LIN {X 0,Y 340.752,Z 249.672,A -85,B 0,C 180,E1 -14239.386,E2 -14239.386} C_VEL
LIN {X 0,Y 341.112,Z 240.977,A -85,B 0,C 180,E1 -14243.046,E2 -14243.046} C_VEL
LIN {X 0,Y 341.383,Z 233.386,A -85,B 0,C 180,E1 -14246.271,E2 -14246.271} C_VEL
LIN {X 0,Y 341.787,Z 224.032,A -85,B 0,C 180,E1 -14250.272,E2 -14250.272} C_VEL
LIN {X 0,Y 342.168,Z 216.106,A -85,B 0,C 180,E1 -14253.681,E2 -14253.681} C_VEL
LIN {X 0,Y 342.261,Z 211.171,A -85,B 0,C 180,E1 -14255.819,E2 -14255.819} C_VEL
LIN {X 0,Y 341.512,Z 205.055,A -85,B 0,C 180,E1 -14258.554,E2 -14258.554} C_VEL
LIN {X 0,Y 340.75,Z 201.041,A -85,B 0,C 180,E1 -14260.45,E2 -14260.45} C_VEL
LIN {X 0,Y 340.658,Z 201.052,A -85,B 0,C 180,E1 -14263.772,E2 -14263.772} C_VEL
LIN {X 0,Y 340.704,Z 201.047,A -85,B 0,C 180,E1 -14267.954,E2 -14267.954} C_VEL
LIN {X 0,Y 340.725,Z 201.046,A -85,B 0,C 180,E1 -14271.77,E2 -14271.77} C_VEL
LIN {X 0,Y 340.727,Z 201.048,A -85,B 0,C 180,E1 -14275.595,E2 -14275.595} C_VEL
LIN {X 0,Y 340.674,Z 201.114,A -85,B 0,C 180,E1 -14278.779,E2 -14278.779} C_VEL
LIN {X 0,Y 340.81,Z 204.268,A -85,B 0,C 180,E1 -14281.685,E2 -14281.685} C_VEL
LIN {X 0,Y 340.762,Z 208.22,A -85,B 0,C 180,E1 -14285.159,E2 -14285.159} C_VEL
LIN {X 0,Y 340.627,Z 211.796,A -85,B 0,C 180,E1 -14288.197,E2 -14288.197} C_VEL
LIN {X 0,Y 340.62,Z 216.505,A -85,B 0,C 180,E1 -14291.97,E2 -14291.97} C_VEL
LIN {X 0,Y 340.593,Z 221.628,A -85,B 0,C 180,E1 -14295.786,E2 -14295.786} C_VEL
LIN {X 0,Y 343.415,Z 232.223,A -85,B 0,C 180,E1 -14296.441,E2 -14296.441} C_VEL
LIN {X 0,Y 345.261,Z 241.478,A -85,B 0,C 180,E1 -14297.204,E2 -14297.204} C_VEL
LIN {X 0,Y 345.073,Z 250.333,A -85,B 0,C 180,E1 -14298.081,E2 -14298.081} C_VEL
LIN {X 0,Y 344.549,Z 257.421,A -85,B 0,C 180,E1 -14298.974,E2 -14298.974} C_VEL
LIN {X 0,Y 343.928,Z 263.871,A -85,B 0,C 180,E1 -14299.996,E2 -14299.996} C_VEL
LIN {X 0,Y 343.24,Z 269.773,A -85,B 0,C 180,E1 -14301.165,E2 -14301.165} C_VEL
LIN {X 0,Y 342.737,Z 274.379,A -85,B 0,C 180,E1 -14302.339,E2 -14302.339} C_VEL
LIN {X 0,Y 342.185,Z 278.047,A -85,B 0,C 180,E1 -14303.512,E2 -14303.512} C_VEL
LIN {X 0,Y 341.789,Z 282.051,A -85,B 0,C 180,E1 -14305.281,E2 -14305.281} C_VEL
LIN {X 0,Y 341.323,Z 283.939,A -85,B 0,C 180,E1 -14306.457,E2 -14306.457} C_VEL
LIN {X 0,Y 341.219,Z 285.215,A -85,B 0,C 180,E1 -14307.638,E2 -14307.638} C_VEL
LIN {X 0,Y 341.059,Z 285.985,A -85,B 0,C 180,E1 -14308.818,E2 -14308.818} C_VEL
LIN {X 0,Y 340.993,Z 286.251,A -85,B 0,C 180,E1 -14309.998,E2 -14309.998} C_VEL
LIN {X 0,Y 341.056,Z 286.023,A -85,B 0,C 180,E1 -14311.179,E2 -14311.179} C_VEL
LIN {X 0,Y 341.213,Z 285.305,A -85,B 0,C 180,E1 -14312.359,E2 -14312.359} C_VEL
LIN {X 0,Y 341.32,Z 284.085,A -85,B 0,C 180,E1 -14313.54,E2 -14313.54} C_VEL
LIN {X 0,Y 342.009,Z 281.111,A -85,B 0,C 180,E1 -14315.304,E2 -14315.304} C_VEL
LIN {X 0,Y 342.279,Z 276.688,A -85,B 0,C 180,E1 -14317.075,E2 -14317.075} C_VEL
LIN {X 0,Y 342.822,Z 273.73,A -85,B 0,C 180,E1 -14317.952,E2 -14317.952} C_VEL
LIN {X 0,Y 343.198,Z 270.243,A -85,B 0,C 180,E1 -14318.833,E2 -14318.833} C_VEL
LIN {X 0,Y 343.922,Z 264.483,A -85,B 0,C 180,E1 -14320.001,E2 -14320.001} C_VEL
LIN {X 0,Y 344.435,Z 259.388,A -85,B 0,C 180,E1 -14320.849,E2 -14320.849} C_VEL
LIN {X 0,Y 344.905,Z 252.666,A -85,B 0,C 180,E1 -14321.756,E2 -14321.756} C_VEL
LIN {X 0,Y 345.44,Z 244.736,A -85,B 0,C 180,E1 -14322.602,E2 -14322.602} C_VEL
LIN {X 0,Y 345.523,Z 242.909,A -85,B 0,C 180,E1 -14322.763,E2 -14322.763} C_VEL
LIN {X 0,Y 343.767,Z 233.855,A -85,B 0,C 180,E1 -14323.547,E2 -14323.547} C_VEL
LIN {X 0,Y 341.183,Z 223.744,A -85,B 0,C 180,E1 -14324.209,E2 -14324.209} C_VEL
LIN {X 0,Y 340.594,Z 221.624,A -85,B 0,C 180,E1 -14324.335,E2 -14324.335} C_VEL
LIN {X 0,Y 340.626,Z 216.247,A -85,B 0,C 180,E1 -14328.359,E2 -14328.359} C_VEL
LIN {X 0,Y 340.65,Z 211.945,A -85,B 0,C 180,E1 -14331.812,E2 -14331.812} C_VEL
LIN {X 0,Y 340.771,Z 207.431,A -85,B 0,C 180,E1 -14335.663,E2 -14335.663} C_VEL
LIN {X 0,Y 340.815,Z 204.47,A -85,B 0,C 180,E1 -14338.311,E2 -14338.311} C_VEL
LIN {X 0,Y 340.696,Z 201.071,A -85,B 0,C 180,E1 -14341.388,E2 -14341.388} C_VEL
LIN {X 0,Y 340.714,Z 201.045,A -85,B 0,C 180,E1 -14345.277,E2 -14345.277} C_VEL
LIN {X 0,Y 340.707,Z 201.045,A -85,B 0,C 180,E1 -14348.385,E2 -14348.385} C_VEL
LIN {X 0,Y 340.693,Z 201.046,A -85,B 0,C 180,E1 -14352.044,E2 -14352.044} C_VEL
LIN {X 0,Y 340.655,Z 201.049,A -85,B 0,C 180,E1 -14353.428,E2 -14353.428} C_VEL
LIN {X 0,Y 339.988,Z 201.133,A -85,B 0,C 180,E1 -14354.413,E2 -14354.413} C_VEL
LIN {X 0,Y 337.121,Z 201.49,A -85,B 0,C 180,E1 -14356.017,E2 -14356.017} C_VEL
LIN {X 0,Y 334.701,Z 201.795,A -85,B 0,C 180,E1 -14357.315,E2 -14357.315} C_VEL
LIN {X 0,Y 333.681,Z 201.921,A -85,B 0,C 180,E1 -14358.32,E2 -14358.32} C_VEL
LIN {X 0,Y 333.607,Z 201.923,A -85,B 0,C 180,E1 -14358.66,E2 -14358.66} C_VEL
LIN {X 0,Y 333.645,Z 201.921,A -85,B 0,C 180,E1 -14362.348,E2 -14362.348} C_VEL
LIN {X 0,Y 333.666,Z 201.919,A -85,B 0,C 180,E1 -14365.34,E2 -14365.34} C_VEL
LIN {X 0,Y 333.691,Z 201.916,A -85,B 0,C 180,E1 -14369.637,E2 -14369.637} C_VEL
LIN {X 0,Y 333.735,Z 201.916,A -85,B 0,C 180,E1 -14372.4,E2 -14372.4} C_VEL
LIN {X 0,Y 333.717,Z 201.905,A -85,B 0,C 180,E1 -14375.09,E2 -14375.09} C_VEL
LIN {X 0,Y 333.672,Z 201.915,A -85,B 0,C 180,E1 -14379.018,E2 -14379.018} C_VEL
LIN {X 0,Y 333.784,Z 201.906,A -85,B 0,C 180,E1 -14381.589,E2 -14381.589} C_VEL
LIN {X 0,Y 333.797,Z 201.897,A -85,B 0,C 180,E1 -14385.576,E2 -14385.576} C_VEL
LIN {X 0,Y 333.823,Z 201.897,A -85,B 0,C 180,E1 -14389.078,E2 -14389.078} C_VEL
LIN {X 0,Y 333.994,Z 201.88,A -85,B 0,C 180,E1 -14392.747,E2 -14392.747} C_VEL
LIN {X 0,Y 333.797,Z 201.895,A -85,B 0,C 180,E1 -14395.169,E2 -14395.169} C_VEL
LIN {X 0,Y 334.095,Z 201.867,A -85,B 0,C 180,E1 -14397.589,E2 -14397.589} C_VEL
LIN {X 0,Y 334.235,Z 201.838,A -85,B 0,C 180,E1 -14400,E2 -14400} C_VEL
LIN {X 0,Y 334.092,Z 201.868,A -85,B 0,C 180,E1 -14402.411,E2 -14402.411} C_VEL
LIN {X 0,Y 334.012,Z 201.878,A -85,B 0,C 180,E1 -14407.253,E2 -14407.253} C_VEL
LIN {X 0,Y 333.822,Z 201.904,A -85,B 0,C 180,E1 -14410.922,E2 -14410.922} C_VEL
LIN {X 0,Y 333.797,Z 201.905,A -85,B 0,C 180,E1 -14414.635,E2 -14414.635} C_VEL
LIN {X 0,Y 333.712,Z 201.917,A -85,B 0,C 180,E1 -14418.618,E2 -14418.618} C_VEL
LIN {X 0,Y 333.64,Z 201.927,A -85,B 0,C 180,E1 -14422.282,E2 -14422.282} C_VEL
LIN {X 0,Y 333.648,Z 201.926,A -85,B 0,C 180,E1 -14425.079,E2 -14425.079} C_VEL
LIN {X 0,Y 333.64,Z 201.927,A -85,B 0,C 180,E1 -14428.979,E2 -14428.979} C_VEL
LIN {X 0,Y 333.634,Z 201.925,A -85,B 0,C 180,E1 -14432.588,E2 -14432.588} C_VEL
LIN {X 0,Y 333.666,Z 201.923,A -85,B 0,C 180,E1 -14436.14,E2 -14436.14} C_VEL
LIN {X 0,Y 333.611,Z 201.927,A -85,B 0,C 180,E1 -14439.197,E2 -14439.197} C_VEL
LIN {X 0,Y 333.621,Z 201.931,A -85,B 0,C 180,E1 -14442.501,E2 -14442.501} C_VEL
LIN {X 0,Y 333.608,Z 201.963,A -85,B 0,C 180,E1 -14445.143,E2 -14445.143} C_VEL
LIN {X 0,Y 335.798,Z 210.783,A -85,B 0,C 180,E1 -14448.891,E2 -14448.891} C_VEL
LIN {X 0,Y 337.805,Z 219.524,A -85,B 0,C 180,E1 -14452.24,E2 -14452.24} C_VEL
LIN {X 0,Y 339.708,Z 228.008,A -85,B 0,C 180,E1 -14455.259,E2 -14455.259} C_VEL
LIN {X 0,Y 340.958,Z 235.046,A -85,B 0,C 180,E1 -14457.595,E2 -14457.595} C_VEL
LIN {X 0,Y 338.442,Z 248.328,A -85,B 0,C 180,E1 -14461.473,E2 -14461.473} C_VEL
LIN {X 0,Y 336.139,Z 262.557,A -85,B 0,C 180,E1 -14465.613,E2 -14465.613} C_VEL
LIN {X 0,Y 334.245,Z 277.674,A -85,B 0,C 180,E1 -14470.043,E2 -14470.043} C_VEL
LIN {X 0,Y 335.25,Z 290.913,A -85,B 0,C 180,E1 -14470.623,E2 -14470.623} C_VEL
LIN {X 0,Y 336.597,Z 313.747,A -85,B 0,C 180,E1 -14472.065,E2 -14472.065} C_VEL
LIN {X 0,Y 336.521,Z 321.792,A -85,B 0,C 180,E1 -14472.688,E2 -14472.688} C_VEL
LIN {X 0,Y 335.458,Z 334.49,A -85,B 0,C 180,E1 -14473.885,E2 -14473.885} C_VEL
LIN {X 0,Y 334.585,Z 345.319,A -85,B 0,C 180,E1 -14475.186,E2 -14475.186} C_VEL
LIN {X 0,Y 333.812,Z 355.01,A -85,B 0,C 180,E1 -14476.611,E2 -14476.611} C_VEL
LIN {X 0,Y 333.237,Z 363.566,A -85,B 0,C 180,E1 -14478.135,E2 -14478.135} C_VEL
LIN {X 0,Y 332.682,Z 371.88,A -85,B 0,C 180,E1 -14479.965,E2 -14479.965} C_VEL
LIN {X 0,Y 332.422,Z 378.567,A -85,B 0,C 180,E1 -14481.797,E2 -14481.797} C_VEL
LIN {X 0,Y 332.288,Z 384.611,A -85,B 0,C 180,E1 -14483.931,E2 -14483.931} C_VEL
LIN {X 0,Y 332.272,Z 388.45,A -85,B 0,C 180,E1 -14485.756,E2 -14485.756} C_VEL
LIN {X 0,Y 332.413,Z 391.197,A -85,B 0,C 180,E1 -14487.578,E2 -14487.578} C_VEL
LIN {X 0,Y 332.392,Z 392.431,A -85,B 0,C 180,E1 -14488.79,E2 -14488.79} C_VEL
LIN {X 0,Y 332.398,Z 393.245,A -85,B 0,C 180,E1 -14490.002,E2 -14490.002} C_VEL
LIN {X 0,Y 332.364,Z 393.606,A -85,B 0,C 180,E1 -14491.213,E2 -14491.213} C_VEL
LIN {X 0,Y 332.207,Z 393.509,A -85,B 0,C 180,E1 -14492.427,E2 -14492.427} C_VEL
LIN {X 0,Y 332.156,Z 393.007,A -85,B 0,C 180,E1 -14493.641,E2 -14493.641} C_VEL
LIN {X 0,Y 332.142,Z 392.099,A -85,B 0,C 180,E1 -14494.857,E2 -14494.857} C_VEL
LIN {X 0,Y 332.153,Z 390.742,A -85,B 0,C 180,E1 -14496.074,E2 -14496.074} C_VEL
LIN {X 0,Y 332.362,Z 387.927,A -85,B 0,C 180,E1 -14497.902,E2 -14497.902} C_VEL
LIN {X 0,Y 332.773,Z 384.115,A -85,B 0,C 180,E1 -14499.729,E2 -14499.729} C_VEL
LIN {X 0,Y 333.487,Z 379.222,A -85,B 0,C 180,E1 -14501.55,E2 -14501.55} C_VEL
LIN {X 0,Y 334.831,Z 372.017,A -85,B 0,C 180,E1 -14503.66,E2 -14503.66} C_VEL
LIN {X 0,Y 336.173,Z 364.432,A -85,B 0,C 180,E1 -14505.461,E2 -14505.461} C_VEL
LIN {X 0,Y 337.605,Z 356.881,A -85,B 0,C 180,E1 -14506.946,E2 -14506.946} C_VEL
LIN {X 0,Y 339.904,Z 345.97,A -85,B 0,C 180,E1 -14508.694,E2 -14508.694} C_VEL
LIN {X 0,Y 342.101,Z 334.974,A -85,B 0,C 180,E1 -14510.129,E2 -14510.129} C_VEL
LIN {X 0,Y 343.964,Z 324.376,A -85,B 0,C 180,E1 -14511.266,E2 -14511.266} C_VEL
LIN {X 0,Y 345.101,Z 311.884,A -85,B 0,C 180,E1 -14512.459,E2 -14512.459} C_VEL
LIN {X 0,Y 345.075,Z 299.035,A -85,B 0,C 180,E1 -14513.58,E2 -14513.58} C_VEL
LIN {X 0,Y 343.453,Z 284.713,A -85,B 0,C 180,E1 -14514.796,E2 -14514.796} C_VEL
LIN {X 0,Y 341.202,Z 273.036,A -85,B 0,C 180,E1 -14515.877,E2 -14515.877} C_VEL
LIN {X 0,Y 341.429,Z 262.711,A -85,B 0,C 180,E1 -14517.734,E2 -14517.734} C_VEL
LIN {X 0,Y 342.068,Z 254.065,A -85,B 0,C 180,E1 -14519.546,E2 -14519.546} C_VEL
LIN {X 0,Y 343.381,Z 244.939,A -85,B 0,C 180,E1 -14521.806,E2 -14521.806} C_VEL
LIN {X 0,Y 344.103,Z 240.547,A -85,B 0,C 180,E1 -14523.134,E2 -14523.134} C_VEL
LIN {X 0,Y 343.908,Z 236.158,A -85,B 0,C 180,E1 -14525.172,E2 -14525.172} C_VEL
LIN {X 0,Y 343.989,Z 232.945,A -85,B 0,C 180,E1 -14527.174,E2 -14527.174} C_VEL
LIN {X 0,Y 344.239,Z 230.518,A -85,B 0,C 180,E1 -14529.266,E2 -14529.266} C_VEL
LIN {X 0,Y 344.234,Z 229.501,A -85,B 0,C 180,E1 -14530.939,E2 -14530.939} C_VEL
LIN {X 0,Y 343.907,Z 229.317,A -85,B 0,C 180,E1 -14532.635,E2 -14532.635} C_VEL
LIN {X 0,Y 343.51,Z 230.306,A -85,B 0,C 180,E1 -14535.923,E2 -14535.923} C_VEL
LIN {X 0,Y 343.392,Z 232.751,A -85,B 0,C 180,E1 -14539.225,E2 -14539.225} C_VEL
LIN {X 0,Y 343.344,Z 235.911,A -85,B 0,C 180,E1 -14542.115,E2 -14542.115} C_VEL
LIN {X 0,Y 343.1,Z 237.846,A -85,B 0,C 180,E1 -14543.556,E2 -14543.556} C_VEL
LIN {X 0,Y 341.056,Z 244.858,A -85,B 0,C 180,E1 -14547.66,E2 -14547.66} C_VEL
LIN {X 0,Y 339.549,Z 252.071,A -85,B 0,C 180,E1 -14551.572,E2 -14551.572} C_VEL
LIN {X 0,Y 338.917,Z 256.838,A -85,B 0,C 180,E1 -14553.975,E2 -14553.975} C_VEL
LIN {X 0,Y 343.148,Z 267.603,A -85,B 0,C 180,E1 -14555.465,E2 -14555.465} C_VEL
LIN {X 0,Y 346.448,Z 278.711,A -85,B 0,C 180,E1 -14556.923,E2 -14556.923} C_VEL
LIN {X 0,Y 347.886,Z 286.492,A -85,B 0,C 180,E1 -14557.908,E2 -14557.908} C_VEL
LIN {X 0,Y 347.59,Z 290.2,A -85,B 0,C 180,E1 -14558.273,E2 -14558.273} C_VEL
LIN {X 0,Y 345.38,Z 302.97,A -85,B 0,C 180,E1 -14559.606,E2 -14559.606} C_VEL
LIN {X 0,Y 343.032,Z 314.829,A -85,B 0,C 180,E1 -14561.175,E2 -14561.175} C_VEL
LIN {X 0,Y 340.728,Z 325.274,A -85,B 0,C 180,E1 -14562.907,E2 -14562.907} C_VEL
LIN {X 0,Y 338.756,Z 333.793,A -85,B 0,C 180,E1 -14564.662,E2 -14564.662} C_VEL
LIN {X 0,Y 337.117,Z 340.723,A -85,B 0,C 180,E1 -14566.436,E2 -14566.436} C_VEL
LIN {X 0,Y 335.629,Z 347.162,A -85,B 0,C 180,E1 -14568.526,E2 -14568.526} C_VEL
LIN {X 0,Y 334.586,Z 351.456,A -85,B 0,C 180,E1 -14570.326,E2 -14570.326} C_VEL
LIN {X 0,Y 334.005,Z 353.755,A -85,B 0,C 180,E1 -14571.53,E2 -14571.53} C_VEL
LIN {X 0,Y 333.364,Z 355.6,A -85,B 0,C 180,E1 -14572.733,E2 -14572.733} C_VEL
LIN {X 0,Y 332.998,Z 358.025,A -85,B 0,C 180,E1 -14575.157,E2 -14575.157} C_VEL
LIN {X 0,Y 332.712,Z 358.621,A -85,B 0,C 180,E1 -14576.367,E2 -14576.367} C_VEL
LIN {X 0,Y 332.318,Z 358.628,A -85,B 0,C 180,E1 -14578.788,E2 -14578.788} C_VEL
LIN {X 0,Y 332.22,Z 358.017,A -85,B 0,C 180,E1 -14580,E2 -14580} C_VEL
LIN {X 0,Y 332.192,Z 356.966,A -85,B 0,C 180,E1 -14581.212,E2 -14581.212} C_VEL
LIN {X 0,Y 332.19,Z 355.515,A -85,B 0,C 180,E1 -14582.425,E2 -14582.425} C_VEL
LIN {X 0,Y 332.318,Z 352.511,A -85,B 0,C 180,E1 -14584.245,E2 -14584.245} C_VEL
LIN {X 0,Y 332.458,Z 348.452,A -85,B 0,C 180,E1 -14586.067,E2 -14586.067} C_VEL
LIN {X 0,Y 332.843,Z 342.227,A -85,B 0,C 180,E1 -14588.194,E2 -14588.194} C_VEL
LIN {X 0,Y 333.379,Z 335.446,A -85,B 0,C 180,E1 -14590.016,E2 -14590.016} C_VEL
LIN {X 0,Y 334.013,Z 327.092,A -85,B 0,C 180,E1 -14591.838,E2 -14591.838} C_VEL
LIN {X 0,Y 334.942,Z 316.687,A -85,B 0,C 180,E1 -14593.654,E2 -14593.654} C_VEL
LIN {X 0,Y 335.846,Z 305.991,A -85,B 0,C 180,E1 -14595.164,E2 -14595.164} C_VEL
LIN {X 0,Y 336.612,Z 294.467,A -85,B 0,C 180,E1 -14596.481,E2 -14596.481} C_VEL
LIN {X 0,Y 337.485,Z 282.446,A -85,B 0,C 180,E1 -14597.575,E2 -14597.575} C_VEL
LIN {X 0,Y 337.858,Z 275.403,A -85,B 0,C 180,E1 -14598.103,E2 -14598.103} C_VEL
LIN {X 0,Y 335.673,Z 262.061,A -85,B 0,C 180,E1 -14599.003,E2 -14599.003} C_VEL
LIN {X 0,Y 333.741,Z 249.961,A -85,B 0,C 180,E1 -14599.633,E2 -14599.633} C_VEL
LIN {X 0,Y 334.135,Z 240.744,A -85,B 0,C 180,E1 -14603.556,E2 -14603.556} C_VEL
LIN {X 0,Y 334.468,Z 231.492,A -85,B 0,C 180,E1 -14607.534,E2 -14607.534} C_VEL
LIN {X 0,Y 334.959,Z 221.997,A -85,B 0,C 180,E1 -14611.638,E2 -14611.638} C_VEL
LIN {X 0,Y 335.281,Z 213.92,A -85,B 0,C 180,E1 -14615.163,E2 -14615.163} C_VEL
LIN {X 0,Y 334.916,Z 208.697,A -85,B 0,C 180,E1 -14617.485,E2 -14617.485} C_VEL
LIN {X 0,Y 333.707,Z 201.919,A -85,B 0,C 180,E1 -14620.644,E2 -14620.644} C_VEL
LIN {X 0,Y 333.599,Z 201.932,A -85,B 0,C 180,E1 -14624.25,E2 -14624.25} C_VEL
LIN {X 0,Y 333.647,Z 201.925,A -85,B 0,C 180,E1 -14627.618,E2 -14627.618} C_VEL
LIN {X 0,Y 333.645,Z 201.927,A -85,B 0,C 180,E1 -14631.204,E2 -14631.204} C_VEL
LIN {X 0,Y 333.678,Z 201.925,A -85,B 0,C 180,E1 -14633.86,E2 -14633.86} C_VEL
LIN {X 0,Y 333.638,Z 201.928,A -85,B 0,C 180,E1 -14637.415,E2 -14637.415} C_VEL
LIN {X 0,Y 333.689,Z 202.166,A -85,B 0,C 180,E1 -14638.581,E2 -14638.581} C_VEL
LIN {X 0,Y 333.797,Z 204.794,A -85,B 0,C 180,E1 -14641.035,E2 -14641.035} C_VEL
LIN {X 0,Y 333.765,Z 207.808,A -85,B 0,C 180,E1 -14643.755,E2 -14643.755} C_VEL
LIN {X 0,Y 333.692,Z 210.874,A -85,B 0,C 180,E1 -14646.41,E2 -14646.41} C_VEL
LIN {X 0,Y 333.578,Z 215.548,A -85,B 0,C 180,E1 -14650.298,E2 -14650.298} C_VEL
LIN {X 0,Y 333.556,Z 218.793,A -85,B 0,C 180,E1 -14652.842,E2 -14652.842} C_VEL
LIN {X 0,Y 333.553,Z 222.253,A -85,B 0,C 180,E1 -14655.411,E2 -14655.411} C_VEL
LIN {X 0,Y 336.552,Z 233.253,A -85,B 0,C 180,E1 -14656.124,E2 -14656.124} C_VEL
LIN {X 0,Y 338.447,Z 242.787,A -85,B 0,C 180,E1 -14656.939,E2 -14656.939} C_VEL
LIN {X 0,Y 338.237,Z 251.449,A -85,B 0,C 180,E1 -14657.829,E2 -14657.829} C_VEL
LIN {X 0,Y 337.667,Z 258.535,A -85,B 0,C 180,E1 -14658.746,E2 -14658.746} C_VEL
LIN {X 0,Y 337.022,Z 264.938,A -85,B 0,C 180,E1 -14659.789,E2 -14659.789} C_VEL
LIN {X 0,Y 336.299,Z 270.802,A -85,B 0,C 180,E1 -14660.981,E2 -14660.981} C_VEL
LIN {X 0,Y 335.775,Z 275.387,A -85,B 0,C 180,E1 -14662.179,E2 -14662.179} C_VEL
LIN {X 0,Y 335.203,Z 279.041,A -85,B 0,C 180,E1 -14663.377,E2 -14663.377} C_VEL
LIN {X 0,Y 334.789,Z 283.032,A -85,B 0,C 180,E1 -14665.182,E2 -14665.182} C_VEL
LIN {X 0,Y 334.311,Z 284.916,A -85,B 0,C 180,E1 -14666.383,E2 -14666.383} C_VEL
LIN {X 0,Y 334.199,Z 286.189,A -85,B 0,C 180,E1 -14667.588,E2 -14667.588} C_VEL
LIN {X 0,Y 334.034,Z 286.959,A -85,B 0,C 180,E1 -14668.793,E2 -14668.793} C_VEL
LIN {X 0,Y 333.966,Z 287.225,A -85,B 0,C 180,E1 -14669.998,E2 -14669.998} C_VEL
LIN {X 0,Y 334.031,Z 286.996,A -85,B 0,C 180,E1 -14671.204,E2 -14671.204} C_VEL
LIN {X 0,Y 334.193,Z 286.279,A -85,B 0,C 180,E1 -14672.409,E2 -14672.409} C_VEL
LIN {X 0,Y 334.308,Z 285.06,A -85,B 0,C 180,E1 -14673.614,E2 -14673.614} C_VEL
LIN {X 0,Y 335.014,Z 282.094,A -85,B 0,C 180,E1 -14675.415,E2 -14675.415} C_VEL
LIN {X 0,Y 335.304,Z 277.685,A -85,B 0,C 180,E1 -14677.223,E2 -14677.223} C_VEL
LIN {X 0,Y 335.865,Z 274.733,A -85,B 0,C 180,E1 -14678.118,E2 -14678.118} C_VEL
LIN {X 0,Y 336.259,Z 271.273,A -85,B 0,C 180,E1 -14679.017,E2 -14679.017} C_VEL
LIN {X 0,Y 337.018,Z 265.544,A -85,B 0,C 180,E1 -14680.208,E2 -14680.208} C_VEL
LIN {X 0,Y 337.558,Z 260.407,A -85,B 0,C 180,E1 -14681.085,E2 -14681.085} C_VEL
LIN {X 0,Y 338.047,Z 253.836,A -85,B 0,C 180,E1 -14681.998,E2 -14681.998} C_VEL
LIN {X 0,Y 338.595,Z 246.012,A -85,B 0,C 180,E1 -14682.861,E2 -14682.861} C_VEL
LIN {X 0,Y 338.415,Z 242.431,A -85,B 0,C 180,E1 -14683.204,E2 -14683.204} C_VEL
LIN {X 0,Y 336.365,Z 232.458,A -85,B 0,C 180,E1 -14684.046,E2 -14684.046} C_VEL
LIN {X 0,Y 333.581,Z 222.227,A -85,B 0,C 180,E1 -14684.721,E2 -14684.721} C_VEL
LIN {X 0,Y 333.605,Z 217.149,A -85,B 0,C 180,E1 -14688.556,E2 -14688.556} C_VEL
LIN {X 0,Y 333.639,Z 212.569,A -85,B 0,C 180,E1 -14692.28,E2 -14692.28} C_VEL
LIN {X 0,Y 333.755,Z 209.259,A -85,B 0,C 180,E1 -14695.113,E2 -14695.113} C_VEL
LIN {X 0,Y 333.847,Z 206.185,A -85,B 0,C 180,E1 -14697.85,E2 -14697.85} C_VEL
LIN {X 0,Y 333.798,Z 203.451,A -85,B 0,C 180,E1 -14700.35,E2 -14700.35} C_VEL
LIN {X 0,Y 333.631,Z 201.927,A -85,B 0,C 180,E1 -14701.914,E2 -14701.914} C_VEL
LIN {X 0,Y 333.681,Z 201.922,A -85,B 0,C 180,E1 -14704.772,E2 -14704.772} C_VEL
LIN {X 0,Y 333.649,Z 201.925,A -85,B 0,C 180,E1 -14707.649,E2 -14707.649} C_VEL
LIN {X 0,Y 333.641,Z 201.927,A -85,B 0,C 180,E1 -14710.766,E2 -14710.766} C_VEL
LIN {X 0,Y 333.619,Z 201.925,A -85,B 0,C 180,E1 -14714.255,E2 -14714.255} C_VEL
LIN {X 0,Y 333.635,Z 201.926,A -85,B 0,C 180,E1 -14717.617,E2 -14717.617} C_VEL
LIN {X 0,Y 333.607,Z 201.923,A -85,B 0,C 180,E1 -14718.66,E2 -14718.66} C_VEL
LIN {X 0,Y 332.963,Z 202.006,A -85,B 0,C 180,E1 -14719.668,E2 -14719.668} C_VEL
LIN {X 0,Y 330.111,Z 202.364,A -85,B 0,C 180,E1 -14721.307,E2 -14721.307} C_VEL
LIN {X 0,Y 327.689,Z 202.662,A -85,B 0,C 180,E1 -14722.634,E2 -14722.634} C_VEL
LIN {X 0,Y 326.662,Z 202.792,A -85,B 0,C 180,E1 -14723.662,E2 -14723.662} C_VEL
LIN {X 0,Y 326.586,Z 202.801,A -85,B 0,C 180,E1 -14724.011,E2 -14724.011} C_VEL
LIN {X 0,Y 326.607,Z 202.799,A -85,B 0,C 180,E1 -14727.455,E2 -14727.455} C_VEL
LIN {X 0,Y 326.653,Z 202.789,A -85,B 0,C 180,E1 -14730.34,E2 -14730.34} C_VEL
LIN {X 0,Y 326.68,Z 202.783,A -85,B 0,C 180,E1 -14734.515,E2 -14734.515} C_VEL
LIN {X 0,Y 326.636,Z 202.793,A -85,B 0,C 180,E1 -14738.544,E2 -14738.544} C_VEL
LIN {X 0,Y 326.734,Z 202.781,A -85,B 0,C 180,E1 -14741.177,E2 -14741.177} C_VEL
LIN {X 0,Y 326.752,Z 202.773,A -85,B 0,C 180,E1 -14745.432,E2 -14745.432} C_VEL
LIN {X 0,Y 326.759,Z 202.779,A -85,B 0,C 180,E1 -14748.838,E2 -14748.838} C_VEL
LIN {X 0,Y 326.946,Z 202.757,A -85,B 0,C 180,E1 -14752.59,E2 -14752.59} C_VEL
LIN {X 0,Y 326.764,Z 202.771,A -85,B 0,C 180,E1 -14755.065,E2 -14755.065} C_VEL
LIN {X 0,Y 327.036,Z 202.747,A -85,B 0,C 180,E1 -14757.537,E2 -14757.537} C_VEL
LIN {X 0,Y 327.187,Z 202.716,A -85,B 0,C 180,E1 -14760,E2 -14760} C_VEL
LIN {X 0,Y 327.032,Z 202.748,A -85,B 0,C 180,E1 -14762.463,E2 -14762.463} C_VEL
LIN {X 0,Y 326.983,Z 202.751,A -85,B 0,C 180,E1 -14766.169,E2 -14766.169} C_VEL
LIN {X 0,Y 326.903,Z 202.758,A -85,B 0,C 180,E1 -14768.655,E2 -14768.655} C_VEL
LIN {X 0,Y 326.723,Z 202.784,A -85,B 0,C 180,E1 -14772.422,E2 -14772.422} C_VEL
LIN {X 0,Y 326.742,Z 202.785,A -85,B 0,C 180,E1 -14774.958,E2 -14774.958} C_VEL
LIN {X 0,Y 326.651,Z 202.797,A -85,B 0,C 180,E1 -14778.828,E2 -14778.828} C_VEL
LIN {X 0,Y 326.581,Z 202.806,A -85,B 0,C 180,E1 -14782.79,E2 -14782.79} C_VEL
LIN {X 0,Y 326.589,Z 202.807,A -85,B 0,C 180,E1 -14785.492,E2 -14785.492} C_VEL
LIN {X 0,Y 326.605,Z 202.804,A -85,B 0,C 180,E1 -14789.665,E2 -14789.665} C_VEL
LIN {X 0,Y 326.607,Z 202.802,A -85,B 0,C 180,E1 -14792.947,E2 -14792.947} C_VEL
LIN {X 0,Y 326.603,Z 202.802,A -85,B 0,C 180,E1 -14795.521,E2 -14795.521} C_VEL
LIN {X 0,Y 326.579,Z 202.803,A -85,B 0,C 180,E1 -14799.223,E2 -14799.223} C_VEL
LIN {X 0,Y 326.566,Z 202.81,A -85,B 0,C 180,E1 -14802.973,E2 -14802.973} C_VEL
LIN {X 0,Y 326.554,Z 202.884,A -85,B 0,C 180,E1 -14804.406,E2 -14804.406} C_VEL
LIN {X 0,Y 328.819,Z 211.988,A -85,B 0,C 180,E1 -14808.424,E2 -14808.424} C_VEL
LIN {X 0,Y 330.791,Z 220.544,A -85,B 0,C 180,E1 -14811.823,E2 -14811.823} C_VEL
LIN {X 0,Y 332.98,Z 230.359,A -85,B 0,C 180,E1 -14815.401,E2 -14815.401} C_VEL
LIN {X 0,Y 334.02,Z 235.953,A -85,B 0,C 180,E1 -14817.312,E2 -14817.312} C_VEL
LIN {X 0,Y 332.864,Z 242.175,A -85,B 0,C 180,E1 -14819.205,E2 -14819.205} C_VEL
LIN {X 0,Y 330.044,Z 257.527,A -85,B 0,C 180,E1 -14823.78,E2 -14823.78} C_VEL
LIN {X 0,Y 327.821,Z 272.432,A -85,B 0,C 180,E1 -14828.298,E2 -14828.298} C_VEL
LIN {X 0,Y 327.273,Z 276.97,A -85,B 0,C 180,E1 -14829.66,E2 -14829.66} C_VEL
LIN {X 0,Y 328.297,Z 289.841,A -85,B 0,C 180,E1 -14830.238,E2 -14830.238} C_VEL
LIN {X 0,Y 328.967,Z 302.224,A -85,B 0,C 180,E1 -14831.048,E2 -14831.048} C_VEL
LIN {X 0,Y 329.623,Z 319.081,A -85,B 0,C 180,E1 -14832.314,E2 -14832.314} C_VEL
LIN {X 0,Y 328.678,Z 330.783,A -85,B 0,C 180,E1 -14833.384,E2 -14833.384} C_VEL
LIN {X 0,Y 327.846,Z 341.908,A -85,B 0,C 180,E1 -14834.666,E2 -14834.666} C_VEL
LIN {X 0,Y 327.062,Z 351.447,A -85,B 0,C 180,E1 -14836.012,E2 -14836.012} C_VEL
LIN {X 0,Y 326.327,Z 360.494,A -85,B 0,C 180,E1 -14837.565,E2 -14837.565} C_VEL
LIN {X 0,Y 325.705,Z 369.332,A -85,B 0,C 180,E1 -14839.433,E2 -14839.433} C_VEL
LIN {X 0,Y 325.418,Z 376.465,A -85,B 0,C 180,E1 -14841.307,E2 -14841.307} C_VEL
LIN {X 0,Y 325.256,Z 382.093,A -85,B 0,C 180,E1 -14843.177,E2 -14843.177} C_VEL
LIN {X 0,Y 325.255,Z 386.46,A -85,B 0,C 180,E1 -14845.043,E2 -14845.043} C_VEL
LIN {X 0,Y 325.184,Z 388.712,A -85,B 0,C 180,E1 -14846.284,E2 -14846.284} C_VEL
LIN {X 0,Y 325.331,Z 390.523,A -85,B 0,C 180,E1 -14847.525,E2 -14847.525} C_VEL
LIN {X 0,Y 325.331,Z 391.816,A -85,B 0,C 180,E1 -14848.764,E2 -14848.764} C_VEL
LIN {X 0,Y 325.334,Z 392.681,A -85,B 0,C 180,E1 -14850.002,E2 -14850.002} C_VEL
LIN {X 0,Y 325.296,Z 393.128,A -85,B 0,C 180,E1 -14851.24,E2 -14851.24} C_VEL
LIN {X 0,Y 325.111,Z 393.11,A -85,B 0,C 180,E1 -14852.479,E2 -14852.479} C_VEL
LIN {X 0,Y 325.075,Z 392.665,A -85,B 0,C 180,E1 -14853.72,E2 -14853.72} C_VEL
LIN {X 0,Y 325.058,Z 390.807,A -85,B 0,C 180,E1 -14855.98,E2 -14855.98} C_VEL
LIN {X 0,Y 325.29,Z 387.862,A -85,B 0,C 180,E1 -14858.075,E2 -14858.075} C_VEL
LIN {X 0,Y 325.761,Z 384.181,A -85,B 0,C 180,E1 -14859.94,E2 -14859.94} C_VEL
LIN {X 0,Y 326.513,Z 379.458,A -85,B 0,C 180,E1 -14861.801,E2 -14861.801} C_VEL
LIN {X 0,Y 327.96,Z 372.481,A -85,B 0,C 180,E1 -14863.952,E2 -14863.952} C_VEL
LIN {X 0,Y 329.637,Z 363.774,A -85,B 0,C 180,E1 -14866.093,E2 -14866.093} C_VEL
LIN {X 0,Y 331.631,Z 354.556,A -85,B 0,C 180,E1 -14867.897,E2 -14867.897} C_VEL
LIN {X 0,Y 334.195,Z 343.367,A -85,B 0,C 180,E1 -14869.664,E2 -14869.664} C_VEL
LIN {X 0,Y 336.601,Z 331.971,A -85,B 0,C 180,E1 -14871.112,E2 -14871.112} C_VEL
LIN {X 0,Y 338.379,Z 321.173,A -85,B 0,C 180,E1 -14872.276,E2 -14872.276} C_VEL
LIN {X 0,Y 339.322,Z 309.133,A -85,B 0,C 180,E1 -14873.446,E2 -14873.446} C_VEL
LIN {X 0,Y 339.147,Z 297.824,A -85,B 0,C 180,E1 -14874.486,E2 -14874.486} C_VEL
LIN {X 0,Y 337.732,Z 285.257,A -85,B 0,C 180,E1 -14875.636,E2 -14875.636} C_VEL
LIN {X 0,Y 335.324,Z 272.573,A -85,B 0,C 180,E1 -14876.91,E2 -14876.91} C_VEL
LIN {X 0,Y 335.866,Z 262.949,A -85,B 0,C 180,E1 -14878.77,E2 -14878.77} C_VEL
LIN {X 0,Y 336.698,Z 254.853,A -85,B 0,C 180,E1 -14880.602,E2 -14880.602} C_VEL
LIN {X 0,Y 338.162,Z 246.829,A -85,B 0,C 180,E1 -14882.709,E2 -14882.709} C_VEL
LIN {X 0,Y 338.533,Z 243.576,A -85,B 0,C 180,E1 -14883.859,E2 -14883.859} C_VEL
LIN {X 0,Y 338.396,Z 239.468,A -85,B 0,C 180,E1 -14885.906,E2 -14885.906} C_VEL
LIN {X 0,Y 338.462,Z 236.462,A -85,B 0,C 180,E1 -14887.903,E2 -14887.903} C_VEL
LIN {X 0,Y 338.564,Z 234.29,A -85,B 0,C 180,E1 -14890.055,E2 -14890.055} C_VEL
LIN {X 0,Y 338.364,Z 233.64,A -85,B 0,C 180,E1 -14891.658,E2 -14891.658} C_VEL
LIN {X 0,Y 338.029,Z 233.595,A -85,B 0,C 180,E1 -14893.324,E2 -14893.324} C_VEL
LIN {X 0,Y 337.531,Z 234.686,A -85,B 0,C 180,E1 -14896.597,E2 -14896.597} C_VEL
LIN {X 0,Y 337.29,Z 237.026,A -85,B 0,C 180,E1 -14899.764,E2 -14899.764} C_VEL
LIN {X 0,Y 337.093,Z 240.27,A -85,B 0,C 180,E1 -14902.799,E2 -14902.799} C_VEL
LIN {X 0,Y 335.611,Z 244.607,A -85,B 0,C 180,E1 -14905.57,E2 -14905.57} C_VEL
LIN {X 0,Y 333.708,Z 251.695,A -85,B 0,C 180,E1 -14909.711,E2 -14909.711} C_VEL
LIN {X 0,Y 332.663,Z 257.53,A -85,B 0,C 180,E1 -14912.834,E2 -14912.834} C_VEL
LIN {X 0,Y 336.421,Z 266.924,A -85,B 0,C 180,E1 -14914.277,E2 -14914.277} C_VEL
LIN {X 0,Y 339.486,Z 276.255,A -85,B 0,C 180,E1 -14915.63,E2 -14915.63} C_VEL
LIN {X 0,Y 341.666,Z 286.178,A -85,B 0,C 180,E1 -14916.994,E2 -14916.994} C_VEL
LIN {X 0,Y 342.026,Z 290.137,A -85,B 0,C 180,E1 -14917.499,E2 -14917.499} C_VEL
LIN {X 0,Y 339.844,Z 302.09,A -85,B 0,C 180,E1 -14918.755,E2 -14918.755} C_VEL
LIN {X 0,Y 337.397,Z 313.555,A -85,B 0,C 180,E1 -14920.25,E2 -14920.25} C_VEL
LIN {X 0,Y 334.96,Z 324.125,A -85,B 0,C 180,E1 -14921.972,E2 -14921.972} C_VEL
LIN {X 0,Y 332.739,Z 332.861,A -85,B 0,C 180,E1 -14923.748,E2 -14923.748} C_VEL
LIN {X 0,Y 330.879,Z 340.047,A -85,B 0,C 180,E1 -14925.548,E2 -14925.548} C_VEL
LIN {X 0,Y 329.231,Z 346.705,A -85,B 0,C 180,E1 -14927.674,E2 -14927.674} C_VEL
LIN {X 0,Y 327.947,Z 351.197,A -85,B 0,C 180,E1 -14929.505,E2 -14929.505} C_VEL
LIN {X 0,Y 327.055,Z 354.629,A -85,B 0,C 180,E1 -14931.349,E2 -14931.349} C_VEL
LIN {X 0,Y 326.373,Z 356.397,A -85,B 0,C 180,E1 -14932.577,E2 -14932.577} C_VEL
LIN {X 0,Y 326.067,Z 357.735,A -85,B 0,C 180,E1 -14933.813,E2 -14933.813} C_VEL
LIN {X 0,Y 325.946,Z 358.631,A -85,B 0,C 180,E1 -14935.052,E2 -14935.052} C_VEL
LIN {X 0,Y 325.657,Z 359.148,A -85,B 0,C 180,E1 -14936.288,E2 -14936.288} C_VEL
LIN {X 0,Y 325.408,Z 359.281,A -85,B 0,C 180,E1 -14937.524,E2 -14937.524} C_VEL
LIN {X 0,Y 325.244,Z 359.008,A -85,B 0,C 180,E1 -14938.762,E2 -14938.762} C_VEL
LIN {X 0,Y 325.095,Z 357.175,A -85,B 0,C 180,E1 -14941.239,E2 -14941.239} C_VEL
LIN {X 0,Y 325.099,Z 355.659,A -85,B 0,C 180,E1 -14942.478,E2 -14942.478} C_VEL
LIN {X 0,Y 325.25,Z 352.527,A -85,B 0,C 180,E1 -14944.337,E2 -14944.337} C_VEL
LIN {X 0,Y 325.413,Z 347.407,A -85,B 0,C 180,E1 -14946.543,E2 -14946.543} C_VEL
LIN {X 0,Y 325.877,Z 340.875,A -85,B 0,C 180,E1 -14948.683,E2 -14948.683} C_VEL
LIN {X 0,Y 326.424,Z 333.667,A -85,B 0,C 180,E1 -14950.545,E2 -14950.545} C_VEL
LIN {X 0,Y 327.13,Z 324.76,A -85,B 0,C 180,E1 -14952.406,E2 -14952.406} C_VEL
LIN {X 0,Y 328.102,Z 314.729,A -85,B 0,C 180,E1 -14954.102,E2 -14954.102} C_VEL
LIN {X 0,Y 329.025,Z 303.21,A -85,B 0,C 180,E1 -14955.683,E2 -14955.683} C_VEL
LIN {X 0,Y 329.921,Z 291.15,A -85,B 0,C 180,E1 -14957,E2 -14957} C_VEL
LIN {X 0,Y 330.807,Z 278.401,A -85,B 0,C 180,E1 -14958.102,E2 -14958.102} C_VEL
LIN {X 0,Y 330.654,Z 275.085,A -85,B 0,C 180,E1 -14958.351,E2 -14958.351} C_VEL
LIN {X 0,Y 328.423,Z 261.33,A -85,B 0,C 180,E1 -14959.279,E2 -14959.279} C_VEL
LIN {X 0,Y 326.675,Z 250.288,A -85,B 0,C 180,E1 -14959.869,E2 -14959.869} C_VEL
LIN {X 0,Y 327.066,Z 242.015,A -85,B 0,C 180,E1 -14963.424,E2 -14963.424} C_VEL
LIN {X 0,Y 327.35,Z 234.24,A -85,B 0,C 180,E1 -14966.799,E2 -14966.799} C_VEL
LIN {X 0,Y 327.738,Z 226.301,A -85,B 0,C 180,E1 -14970.261,E2 -14970.261} C_VEL
LIN {X 0,Y 328.181,Z 218.159,A -85,B 0,C 180,E1 -14973.834,E2 -14973.834} C_VEL
LIN {X 0,Y 328.239,Z 212.999,A -85,B 0,C 180,E1 -14976.131,E2 -14976.131} C_VEL
LIN {X 0,Y 327.602,Z 207.852,A -85,B 0,C 180,E1 -14978.472,E2 -14978.472} C_VEL
LIN {X 0,Y 326.664,Z 202.796,A -85,B 0,C 180,E1 -14980.925,E2 -14980.925} C_VEL
LIN {X 0,Y 326.533,Z 202.808,A -85,B 0,C 180,E1 -14984.742,E2 -14984.742} C_VEL
LIN {X 0,Y 326.581,Z 202.806,A -85,B 0,C 180,E1 -14988.153,E2 -14988.153} C_VEL
LIN {X 0,Y 326.592,Z 202.807,A -85,B 0,C 180,E1 -14991.385,E2 -14991.385} C_VEL
LIN {X 0,Y 326.623,Z 202.804,A -85,B 0,C 180,E1 -14994.851,E2 -14994.851} C_VEL
LIN {X 0,Y 326.603,Z 202.843,A -85,B 0,C 180,E1 -14998,E2 -14998} C_VEL
LIN {X 0,Y 326.809,Z 205.311,A -85,B 0,C 180,E1 -15000.354,E2 -15000.354} C_VEL
LIN {X 0,Y 326.793,Z 208.379,A -85,B 0,C 180,E1 -15003.15,E2 -15003.15} C_VEL
LIN {X 0,Y 326.709,Z 211.452,A -85,B 0,C 180,E1 -15005.874,E2 -15005.874} C_VEL
LIN {X 0,Y 326.586,Z 216.199,A -85,B 0,C 180,E1 -15009.859,E2 -15009.859} C_VEL
LIN {X 0,Y 326.55,Z 219.477,A -85,B 0,C 180,E1 -15012.462,E2 -15012.462} C_VEL
LIN {X 0,Y 326.545,Z 222.888,A -85,B 0,C 180,E1 -15015.031,E2 -15015.031} C_VEL
LIN {X 0,Y 329.58,Z 233.783,A -85,B 0,C 180,E1 -15015.754,E2 -15015.754} C_VEL
LIN {X 0,Y 331.396,Z 242.493,A -85,B 0,C 180,E1 -15016.508,E2 -15016.508} C_VEL
LIN {X 0,Y 331.801,Z 245.451,A -85,B 0,C 180,E1 -15016.812,E2 -15016.812} C_VEL
LIN {X 0,Y 331.341,Z 253.288,A -85,B 0,C 180,E1 -15017.654,E2 -15017.654} C_VEL
LIN {X 0,Y 330.8,Z 259.645,A -85,B 0,C 180,E1 -15018.51,E2 -15018.51} C_VEL
LIN {X 0,Y 330.121,Z 266.003,A -85,B 0,C 180,E1 -15019.573,E2 -15019.573} C_VEL
LIN {X 0,Y 329.36,Z 271.83,A -85,B 0,C 180,E1 -15020.789,E2 -15020.789} C_VEL
LIN {X 0,Y 328.815,Z 276.394,A -85,B 0,C 180,E1 -15022.013,E2 -15022.013} C_VEL
LIN {X 0,Y 328.224,Z 280.035,A -85,B 0,C 180,E1 -15023.235,E2 -15023.235} C_VEL
LIN {X 0,Y 327.789,Z 284.012,A -85,B 0,C 180,E1 -15025.079,E2 -15025.079} C_VEL
LIN {X 0,Y 327.299,Z 285.892,A -85,B 0,C 180,E1 -15026.305,E2 -15026.305} C_VEL
LIN {X 0,Y 327.18,Z 287.163,A -85,B 0,C 180,E1 -15027.536,E2 -15027.536} C_VEL
LIN {X 0,Y 327.009,Z 287.933,A -85,B 0,C 180,E1 -15028.767,E2 -15028.767} C_VEL
LIN {X 0,Y 326.94,Z 288.199,A -85,B 0,C 180,E1 -15029.998,E2 -15029.998} C_VEL
LIN {X 0,Y 327.007,Z 287.97,A -85,B 0,C 180,E1 -15031.23,E2 -15031.23} C_VEL
LIN {X 0,Y 327.174,Z 287.253,A -85,B 0,C 180,E1 -15032.461,E2 -15032.461} C_VEL
LIN {X 0,Y 327.296,Z 286.036,A -85,B 0,C 180,E1 -15033.692,E2 -15033.692} C_VEL
LIN {X 0,Y 328.02,Z 283.076,A -85,B 0,C 180,E1 -15035.531,E2 -15035.531} C_VEL
LIN {X 0,Y 328.332,Z 278.681,A -85,B 0,C 180,E1 -15037.377,E2 -15037.377} C_VEL
LIN {X 0,Y 328.91,Z 275.736,A -85,B 0,C 180,E1 -15038.291,E2 -15038.291} C_VEL
LIN {X 0,Y 329.324,Z 272.3,A -85,B 0,C 180,E1 -15039.208,E2 -15039.208} C_VEL
LIN {X 0,Y 330.117,Z 266.604,A -85,B 0,C 180,E1 -15040.424,E2 -15040.424} C_VEL
LIN {X 0,Y 330.856,Z 259.524,A -85,B 0,C 180,E1 -15041.616,E2 -15041.616} C_VEL
LIN {X 0,Y 331.355,Z 252.504,A -85,B 0,C 180,E1 -15042.555,E2 -15042.555} C_VEL
LIN {X 0,Y 331.868,Z 245.338,A -85,B 0,C 180,E1 -15043.313,E2 -15043.313} C_VEL
LIN {X 0,Y 329.988,Z 235.548,A -85,B 0,C 180,E1 -15044.219,E2 -15044.219} C_VEL
LIN {X 0,Y 327.197,Z 225.168,A -85,B 0,C 180,E1 -15044.948,E2 -15044.948} C_VEL
LIN {X 0,Y 326.579,Z 222.892,A -85,B 0,C 180,E1 -15045.084,E2 -15045.084} C_VEL
LIN {X 0,Y 326.595,Z 217.99,A -85,B 0,C 180,E1 -15048.83,E2 -15048.83} C_VEL
LIN {X 0,Y 326.653,Z 213.192,A -85,B 0,C 180,E1 -15052.783,E2 -15052.783} C_VEL
LIN {X 0,Y 326.776,Z 210.057,A -85,B 0,C 180,E1 -15055.475,E2 -15055.475} C_VEL
LIN {X 0,Y 326.848,Z 207.055,A -85,B 0,C 180,E1 -15058.23,E2 -15058.23} C_VEL
LIN {X 0,Y 326.678,Z 203.182,A -85,B 0,C 180,E1 -15061.806,E2 -15061.806} C_VEL
LIN {X 0,Y 326.595,Z 202.803,A -85,B 0,C 180,E1 -15062.544,E2 -15062.544} C_VEL
LIN {X 0,Y 326.609,Z 202.803,A -85,B 0,C 180,E1 -15065.518,E2 -15065.518} C_VEL
LIN {X 0,Y 326.607,Z 202.803,A -85,B 0,C 180,E1 -15069.226,E2 -15069.226} C_VEL
LIN {X 0,Y 326.576,Z 202.808,A -85,B 0,C 180,E1 -15072.971,E2 -15072.971} C_VEL
LIN {X 0,Y 326.575,Z 202.804,A -85,B 0,C 180,E1 -15077.025,E2 -15077.025} C_VEL
LIN {X 0,Y 326.604,Z 202.803,A -85,B 0,C 180,E1 -15080.771,E2 -15080.771} C_VEL
LIN {X 0,Y 326.586,Z 202.801,A -85,B 0,C 180,E1 -15084.011,E2 -15084.011} C_VEL
LIN {X 0,Y 325.932,Z 202.888,A -85,B 0,C 180,E1 -15085.039,E2 -15085.039} C_VEL
LIN {X 0,Y 323.069,Z 203.245,A -85,B 0,C 180,E1 -15086.712,E2 -15086.712} C_VEL
LIN {X 0,Y 320.653,Z 203.543,A -85,B 0,C 180,E1 -15088.068,E2 -15088.068} C_VEL
LIN {X 0,Y 319.644,Z 203.667,A -85,B 0,C 180,E1 -15089.119,E2 -15089.119} C_VEL
LIN {X 0,Y 319.577,Z 203.674,A -85,B 0,C 180,E1 -15089.474,E2 -15089.474} C_VEL
LIN {X 0,Y 319.6,Z 203.676,A -85,B 0,C 180,E1 -15092.497,E2 -15092.497} C_VEL
LIN {X 0,Y 319.595,Z 203.664,A -85,B 0,C 180,E1 -15095.303,E2 -15095.303} C_VEL
LIN {X 0,Y 319.587,Z 203.674,A -85,B 0,C 180,E1 -15098.047,E2 -15098.047} C_VEL
LIN {X 0,Y 319.679,Z 203.659,A -85,B 0,C 180,E1 -15100.961,E2 -15100.961} C_VEL
LIN {X 0,Y 319.72,Z 203.647,A -85,B 0,C 180,E1 -15105.275,E2 -15105.275} C_VEL
LIN {X 0,Y 319.742,Z 203.644,A -85,B 0,C 180,E1 -15109.872,E2 -15109.872} C_VEL
LIN {X 0,Y 319.901,Z 203.634,A -85,B 0,C 180,E1 -15112.425,E2 -15112.425} C_VEL
LIN {X 0,Y 319.733,Z 203.647,A -85,B 0,C 180,E1 -15114.956,E2 -15114.956} C_VEL
LIN {X 0,Y 319.98,Z 203.626,A -85,B 0,C 180,E1 -15117.482,E2 -15117.482} C_VEL
LIN {X 0,Y 320.138,Z 203.594,A -85,B 0,C 180,E1 -15120,E2 -15120} C_VEL
LIN {X 0,Y 319.976,Z 203.627,A -85,B 0,C 180,E1 -15122.518,E2 -15122.518} C_VEL
LIN {X 0,Y 319.938,Z 203.629,A -85,B 0,C 180,E1 -15126.306,E2 -15126.306} C_VEL
LIN {X 0,Y 319.831,Z 203.637,A -85,B 0,C 180,E1 -15128.848,E2 -15128.848} C_VEL
LIN {X 0,Y 319.67,Z 203.659,A -85,B 0,C 180,E1 -15132.7,E2 -15132.7} C_VEL
LIN {X 0,Y 319.672,Z 203.665,A -85,B 0,C 180,E1 -15135.297,E2 -15135.297} C_VEL
LIN {X 0,Y 319.576,Z 203.678,A -85,B 0,C 180,E1 -15139.261,E2 -15139.261} C_VEL
LIN {X 0,Y 319.531,Z 203.685,A -85,B 0,C 180,E1 -15143.322,E2 -15143.322} C_VEL
LIN {X 0,Y 319.539,Z 203.684,A -85,B 0,C 180,E1 -15146.097,E2 -15146.097} C_VEL
LIN {X 0,Y 319.531,Z 203.685,A -85,B 0,C 180,E1 -15148.939,E2 -15148.939} C_VEL
LIN {X 0,Y 319.514,Z 203.686,A -85,B 0,C 180,E1 -15151.864,E2 -15151.864} C_VEL
LIN {X 0,Y 319.57,Z 203.678,A -85,B 0,C 180,E1 -15155.544,E2 -15155.544} C_VEL
LIN {X 0,Y 319.519,Z 203.675,A -85,B 0,C 180,E1 -15159.663,E2 -15159.663} C_VEL
LIN {X 0,Y 319.541,Z 203.872,A -85,B 0,C 180,E1 -15163.696,E2 -15163.696} C_VEL
LIN {X 0,Y 321.484,Z 211.792,A -85,B 0,C 180,E1 -15167.339,E2 -15167.339} C_VEL
LIN {X 0,Y 323.175,Z 218.811,A -85,B 0,C 180,E1 -15170.296,E2 -15170.296} C_VEL
LIN {X 0,Y 325.193,Z 227.787,A -85,B 0,C 180,E1 -15173.767,E2 -15173.767} C_VEL
LIN {X 0,Y 326.988,Z 236.664,A -85,B 0,C 180,E1 -15176.954,E2 -15176.954} C_VEL
LIN {X 0,Y 326.755,Z 239.433,A -85,B 0,C 180,E1 -15177.839,E2 -15177.839} C_VEL
LIN {X 0,Y 324.04,Z 252.487,A -85,B 0,C 180,E1 -15181.856,E2 -15181.856} C_VEL
LIN {X 0,Y 321.647,Z 266.608,A -85,B 0,C 180,E1 -15186.228,E2 -15186.228} C_VEL
LIN {X 0,Y 320.332,Z 276.272,A -85,B 0,C 180,E1 -15189.262,E2 -15189.262} C_VEL
LIN {X 0,Y 321.359,Z 288.867,A -85,B 0,C 180,E1 -15189.841,E2 -15189.841} C_VEL
LIN {X 0,Y 321.946,Z 301.24,A -85,B 0,C 180,E1 -15190.661,E2 -15190.661} C_VEL
LIN {X 0,Y 322.571,Z 318.011,A -85,B 0,C 180,E1 -15192.078,E2 -15192.078} C_VEL
LIN {X 0,Y 321.864,Z 328.343,A -85,B 0,C 180,E1 -15193.021,E2 -15193.021} C_VEL
LIN {X 0,Y 320.984,Z 339.475,A -85,B 0,C 180,E1 -15194.282,E2 -15194.282} C_VEL
LIN {X 0,Y 320.074,Z 349.716,A -85,B 0,C 180,E1 -15195.716,E2 -15195.716} C_VEL
LIN {X 0,Y 319.333,Z 358.94,A -85,B 0,C 180,E1 -15197.288,E2 -15197.288} C_VEL
LIN {X 0,Y 318.765,Z 366.638,A -85,B 0,C 180,E1 -15198.879,E2 -15198.879} C_VEL
LIN {X 0,Y 318.394,Z 374.164,A -85,B 0,C 180,E1 -15200.793,E2 -15200.793} C_VEL
LIN {X 0,Y 318.188,Z 381.085,A -85,B 0,C 180,E1 -15203.024,E2 -15203.024} C_VEL
LIN {X 0,Y 318.189,Z 385.592,A -85,B 0,C 180,E1 -15204.933,E2 -15204.933} C_VEL
LIN {X 0,Y 318.115,Z 387.908,A -85,B 0,C 180,E1 -15206.201,E2 -15206.201} C_VEL
LIN {X 0,Y 318.251,Z 389.788,A -85,B 0,C 180,E1 -15207.47,E2 -15207.47} C_VEL
LIN {X 0,Y 318.27,Z 391.189,A -85,B 0,C 180,E1 -15208.736,E2 -15208.736} C_VEL
LIN {X 0,Y 318.27,Z 392.109,A -85,B 0,C 180,E1 -15210.002,E2 -15210.002} C_VEL
LIN {X 0,Y 318.229,Z 392.611,A -85,B 0,C 180,E1 -15211.267,E2 -15211.267} C_VEL
LIN {X 0,Y 318.017,Z 392.689,A -85,B 0,C 180,E1 -15212.535,E2 -15212.535} C_VEL
LIN {X 0,Y 317.996,Z 392.327,A -85,B 0,C 180,E1 -15213.803,E2 -15213.803} C_VEL
LIN {X 0,Y 317.977,Z 390.762,A -85,B 0,C 180,E1 -15215.954,E2 -15215.954} C_VEL
LIN {X 0,Y 318.231,Z 387.784,A -85,B 0,C 180,E1 -15218.255,E2 -15218.255} C_VEL
LIN {X 0,Y 318.746,Z 384.249,A -85,B 0,C 180,E1 -15220.161,E2 -15220.161} C_VEL
LIN {X 0,Y 319.557,Z 379.7,A -85,B 0,C 180,E1 -15222.061,E2 -15222.061} C_VEL
LIN {X 0,Y 321.101,Z 372.991,A -85,B 0,C 180,E1 -15224.256,E2 -15224.256} C_VEL
LIN {X 0,Y 322.858,Z 364.538,A -85,B 0,C 180,E1 -15226.44,E2 -15226.44} C_VEL
LIN {X 0,Y 324.965,Z 355.7,A -85,B 0,C 180,E1 -15228.277,E2 -15228.277} C_VEL
LIN {X 0,Y 327.647,Z 344.911,A -85,B 0,C 180,E1 -15230.073,E2 -15230.073} C_VEL
LIN {X 0,Y 330.147,Z 334.124,A -85,B 0,C 180,E1 -15231.545,E2 -15231.545} C_VEL
LIN {X 0,Y 331.896,Z 325.236,A -85,B 0,C 180,E1 -15232.571,E2 -15232.571} C_VEL
LIN {X 0,Y 333.313,Z 313.513,A -85,B 0,C 180,E1 -15233.8,E2 -15233.8} C_VEL
LIN {X 0,Y 333.654,Z 302.128,A -85,B 0,C 180,E1 -15234.917,E2 -15234.917} C_VEL
LIN {X 0,Y 332.764,Z 290.127,A -85,B 0,C 180,E1 -15236.097,E2 -15236.097} C_VEL
LIN {X 0,Y 331.001,Z 278.971,A -85,B 0,C 180,E1 -15237.231,E2 -15237.231} C_VEL
LIN {X 0,Y 329.676,Z 271.902,A -85,B 0,C 180,E1 -15238.052,E2 -15238.052} C_VEL
LIN {X 0,Y 330.684,Z 261.282,A -85,B 0,C 180,E1 -15240.317,E2 -15240.317} C_VEL
LIN {X 0,Y 332.187,Z 252.203,A -85,B 0,C 180,E1 -15242.65,E2 -15242.65} C_VEL
LIN {X 0,Y 332.724,Z 249.931,A -85,B 0,C 180,E1 -15243.313,E2 -15243.313} C_VEL
LIN {X 0,Y 332.94,Z 248.178,A -85,B 0,C 180,E1 -15243.934,E2 -15243.934} C_VEL
LIN {X 0,Y 332.862,Z 245.13,A -85,B 0,C 180,E1 -15245.346,E2 -15245.346} C_VEL
LIN {X 0,Y 332.862,Z 241.174,A -85,B 0,C 180,E1 -15247.758,E2 -15247.758} C_VEL
LIN {X 0,Y 332.932,Z 239.384,A -85,B 0,C 180,E1 -15249.294,E2 -15249.294} C_VEL
LIN {X 0,Y 332.797,Z 238.263,A -85,B 0,C 180,E1 -15250.895,E2 -15250.895} C_VEL
LIN {X 0,Y 332.436,Z 237.818,A -85,B 0,C 180,E1 -15252.573,E2 -15252.573} C_VEL
LIN {X 0,Y 331.772,Z 238.285,A -85,B 0,C 180,E1 -15255.649,E2 -15255.649} C_VEL
LIN {X 0,Y 331.313,Z 240.096,A -85,B 0,C 180,E1 -15258.884,E2 -15258.884} C_VEL
LIN {X 0,Y 331.017,Z 242.715,A -85,B 0,C 180,E1 -15261.775,E2 -15261.775} C_VEL
LIN {X 0,Y 330.204,Z 245.563,A -85,B 0,C 180,E1 -15263.979,E2 -15263.979} C_VEL
LIN {X 0,Y 327.859,Z 252.509,A -85,B 0,C 180,E1 -15268.319,E2 -15268.319} C_VEL
LIN {X 0,Y 326.559,Z 258.353,A -85,B 0,C 180,E1 -15271.587,E2 -15271.587} C_VEL
LIN {X 0,Y 331.143,Z 269.64,A -85,B 0,C 180,E1 -15273.532,E2 -15273.532} C_VEL
LIN {X 0,Y 334.401,Z 280.708,A -85,B 0,C 180,E1 -15275.235,E2 -15275.235} C_VEL
LIN {X 0,Y 336.131,Z 289.986,A -85,B 0,C 180,E1 -15276.593,E2 -15276.593} C_VEL
LIN {X 0,Y 336.247,Z 292.082,A -85,B 0,C 180,E1 -15276.879,E2 -15276.879} C_VEL
LIN {X 0,Y 334.037,Z 303.138,A -85,B 0,C 180,E1 -15278.079,E2 -15278.079} C_VEL
LIN {X 0,Y 331.546,Z 313.969,A -85,B 0,C 180,E1 -15279.527,E2 -15279.527} C_VEL
LIN {X 0,Y 328.917,Z 324.65,A -85,B 0,C 180,E1 -15281.306,E2 -15281.306} C_VEL
LIN {X 0,Y 326.486,Z 333.347,A -85,B 0,C 180,E1 -15283.106,E2 -15283.106} C_VEL
LIN {X 0,Y 324.489,Z 340.491,A -85,B 0,C 180,E1 -15284.936,E2 -15284.936} C_VEL
LIN {X 0,Y 322.907,Z 346.298,A -85,B 0,C 180,E1 -15286.789,E2 -15286.789} C_VEL
LIN {X 0,Y 321.511,Z 350.963,A -85,B 0,C 180,E1 -15288.654,E2 -15288.654} C_VEL
LIN {X 0,Y 320.179,Z 355.336,A -85,B 0,C 180,E1 -15291.033,E2 -15291.033} C_VEL
LIN {X 0,Y 319.385,Z 357.216,A -85,B 0,C 180,E1 -15292.413,E2 -15292.413} C_VEL
LIN {X 0,Y 319.033,Z 358.432,A -85,B 0,C 180,E1 -15293.676,E2 -15293.676} C_VEL
LIN {X 0,Y 318.898,Z 359.237,A -85,B 0,C 180,E1 -15294.943,E2 -15294.943} C_VEL
LIN {X 0,Y 318.604,Z 359.68,A -85,B 0,C 180,E1 -15296.206,E2 -15296.206} C_VEL
LIN {X 0,Y 318.328,Z 359.734,A -85,B 0,C 180,E1 -15297.469,E2 -15297.469} C_VEL
LIN {X 0,Y 318.154,Z 359.341,A -85,B 0,C 180,E1 -15298.734,E2 -15298.734} C_VEL
LIN {X 0,Y 317.998,Z 357.371,A -85,B 0,C 180,E1 -15301.266,E2 -15301.266} C_VEL
LIN {X 0,Y 318.045,Z 354.769,A -85,B 0,C 180,E1 -15303.167,E2 -15303.167} C_VEL
LIN {X 0,Y 318.213,Z 351.157,A -85,B 0,C 180,E1 -15305.068,E2 -15305.068} C_VEL
LIN {X 0,Y 318.511,Z 345.224,A -85,B 0,C 180,E1 -15307.389,E2 -15307.389} C_VEL
LIN {X 0,Y 319.002,Z 338.192,A -85,B 0,C 180,E1 -15309.511,E2 -15309.511} C_VEL
LIN {X 0,Y 319.654,Z 330.237,A -85,B 0,C 180,E1 -15311.413,E2 -15311.413} C_VEL
LIN {X 0,Y 320.493,Z 320.459,A -85,B 0,C 180,E1 -15313.312,E2 -15313.312} C_VEL
LIN {X 0,Y 321.334,Z 310.413,A -85,B 0,C 180,E1 -15314.892,E2 -15314.892} C_VEL
LIN {X 0,Y 322.091,Z 301.288,A -85,B 0,C 180,E1 -15316.088,E2 -15316.088} C_VEL
LIN {X 0,Y 323.079,Z 289.045,A -85,B 0,C 180,E1 -15317.404,E2 -15317.404} C_VEL
LIN {X 0,Y 323.81,Z 276.935,A -85,B 0,C 180,E1 -15318.425,E2 -15318.425} C_VEL
LIN {X 0,Y 321.576,Z 263.147,A -85,B 0,C 180,E1 -15319.412,E2 -15319.412} C_VEL
LIN {X 0,Y 319.651,Z 250.615,A -85,B 0,C 180,E1 -15320.104,E2 -15320.104} C_VEL
LIN {X 0,Y 320.093,Z 241.722,A -85,B 0,C 180,E1 -15323.966,E2 -15323.966} C_VEL
LIN {X 0,Y 320.406,Z 233.837,A -85,B 0,C 180,E1 -15327.428,E2 -15327.428} C_VEL
LIN {X 0,Y 320.931,Z 224.152,A -85,B 0,C 180,E1 -15331.707,E2 -15331.707} C_VEL
LIN {X 0,Y 321.275,Z 216.08,A -85,B 0,C 180,E1 -15335.306,E2 -15335.306} C_VEL
LIN {X 0,Y 320.875,Z 210.547,A -85,B 0,C 180,E1 -15337.827,E2 -15337.827} C_VEL
LIN {X 0,Y 319.582,Z 203.679,A -85,B 0,C 180,E1 -15341.085,E2 -15341.085} C_VEL
LIN {X 0,Y 319.494,Z 203.685,A -85,B 0,C 180,E1 -15344.742,E2 -15344.742} C_VEL
LIN {X 0,Y 319.53,Z 203.684,A -85,B 0,C 180,E1 -15348.403,E2 -15348.403} C_VEL
LIN {X 0,Y 319.54,Z 203.686,A -85,B 0,C 180,E1 -15351.986,E2 -15351.986} C_VEL
LIN {X 0,Y 319.563,Z 203.683,A -85,B 0,C 180,E1 -15355.122,E2 -15355.122} C_VEL
LIN {X 0,Y 319.575,Z 203.742,A -85,B 0,C 180,E1 -15357.583,E2 -15357.583} C_VEL
LIN {X 0,Y 319.825,Z 205.843,A -85,B 0,C 180,E1 -15359.64,E2 -15359.64} C_VEL
LIN {X 0,Y 319.809,Z 208.934,A -85,B 0,C 180,E1 -15362.515,E2 -15362.515} C_VEL
LIN {X 0,Y 319.733,Z 212.064,A -85,B 0,C 180,E1 -15365.313,E2 -15365.313} C_VEL
LIN {X 0,Y 319.603,Z 215.225,A -85,B 0,C 180,E1 -15368.047,E2 -15368.047} C_VEL
LIN {X 0,Y 319.601,Z 218.82,A -85,B 0,C 180,E1 -15371.009,E2 -15371.009} C_VEL
LIN {X 0,Y 319.543,Z 223.69,A -85,B 0,C 180,E1 -15374.644,E2 -15374.644} C_VEL
LIN {X 0,Y 322.478,Z 234.021,A -85,B 0,C 180,E1 -15375.339,E2 -15375.339} C_VEL
LIN {X 0,Y 324.61,Z 243.858,A -85,B 0,C 180,E1 -15376.221,E2 -15376.221} C_VEL
LIN {X 0,Y 325.002,Z 246.661,A -85,B 0,C 180,E1 -15376.525,E2 -15376.525} C_VEL
LIN {X 0,Y 324.504,Z 254.271,A -85,B 0,C 180,E1 -15377.364,E2 -15377.364} C_VEL
LIN {X 0,Y 323.933,Z 260.756,A -85,B 0,C 180,E1 -15378.263,E2 -15378.263} C_VEL
LIN {X 0,Y 323.224,Z 267.068,A -85,B 0,C 180,E1 -15379.348,E2 -15379.348} C_VEL
LIN {X 0,Y 322.426,Z 272.857,A -85,B 0,C 180,E1 -15380.59,E2 -15380.59} C_VEL
LIN {X 0,Y 321.859,Z 277.401,A -85,B 0,C 180,E1 -15381.839,E2 -15381.839} C_VEL
LIN {X 0,Y 321.246,Z 281.028,A -85,B 0,C 180,E1 -15383.088,E2 -15383.088} C_VEL
LIN {X 0,Y 320.791,Z 284.993,A -85,B 0,C 180,E1 -15384.971,E2 -15384.971} C_VEL
LIN {X 0,Y 320.288,Z 286.869,A -85,B 0,C 180,E1 -15386.224,E2 -15386.224} C_VEL
LIN {X 0,Y 320.16,Z 288.138,A -85,B 0,C 180,E1 -15387.482,E2 -15387.482} C_VEL
LIN {X 0,Y 319.985,Z 288.906,A -85,B 0,C 180,E1 -15388.74,E2 -15388.74} C_VEL
LIN {X 0,Y 319.913,Z 289.173,A -85,B 0,C 180,E1 -15389.998,E2 -15389.998} C_VEL
LIN {X 0,Y 319.982,Z 288.943,A -85,B 0,C 180,E1 -15391.257,E2 -15391.257} C_VEL
LIN {X 0,Y 320.155,Z 288.226,A -85,B 0,C 180,E1 -15392.515,E2 -15392.515} C_VEL
LIN {X 0,Y 320.285,Z 287.011,A -85,B 0,C 180,E1 -15393.773,E2 -15393.773} C_VEL
LIN {X 0,Y 321.026,Z 284.058,A -85,B 0,C 180,E1 -15395.652,E2 -15395.652} C_VEL
LIN {X 0,Y 321.363,Z 279.675,A -85,B 0,C 180,E1 -15397.538,E2 -15397.538} C_VEL
LIN {X 0,Y 321.958,Z 276.739,A -85,B 0,C 180,E1 -15398.471,E2 -15398.471} C_VEL
LIN {X 0,Y 322.393,Z 273.324,A -85,B 0,C 180,E1 -15399.408,E2 -15399.408} C_VEL
LIN {X 0,Y 323.22,Z 267.663,A -85,B 0,C 180,E1 -15400.649,E2 -15400.649} C_VEL
LIN {X 0,Y 324.006,Z 260.565,A -85,B 0,C 180,E1 -15401.875,E2 -15401.875} C_VEL
LIN {X 0,Y 324.491,Z 253.924,A -85,B 0,C 180,E1 -15402.793,E2 -15402.793} C_VEL
LIN {X 0,Y 325.034,Z 246.798,A -85,B 0,C 180,E1 -15403.582,E2 -15403.582} C_VEL
LIN {X 0,Y 323.321,Z 237.454,A -85,B 0,C 180,E1 -15404.49,E2 -15404.49} C_VEL
LIN {X 0,Y 320.546,Z 227.053,A -85,B 0,C 180,E1 -15405.267,E2 -15405.267} C_VEL
LIN {X 0,Y 319.596,Z 223.527,A -85,B 0,C 180,E1 -15405.482,E2 -15405.482} C_VEL
LIN {X 0,Y 319.601,Z 218.655,A -85,B 0,C 180,E1 -15409.258,E2 -15409.258} C_VEL
LIN {X 0,Y 319.656,Z 213.797,A -85,B 0,C 180,E1 -15413.311,E2 -15413.311} C_VEL
LIN {X 0,Y 319.797,Z 210.646,A -85,B 0,C 180,E1 -15416.072,E2 -15416.072} C_VEL
LIN {X 0,Y 319.835,Z 207.587,A -85,B 0,C 180,E1 -15418.907,E2 -15418.907} C_VEL
LIN {X 0,Y 319.708,Z 204.464,A -85,B 0,C 180,E1 -15421.84,E2 -15421.84} C_VEL
LIN {X 0,Y 319.554,Z 203.681,A -85,B 0,C 180,E1 -15422.779,E2 -15422.779} C_VEL
LIN {X 0,Y 319.555,Z 203.679,A -85,B 0,C 180,E1 -15426.426,E2 -15426.426} C_VEL
LIN {X 0,Y 319.553,Z 203.68,A -85,B 0,C 180,E1 -15429.667,E2 -15429.667} C_VEL
LIN {X 0,Y 319.551,Z 203.678,A -85,B 0,C 180,E1 -15433.466,E2 -15433.466} C_VEL
LIN {X 0,Y 319.554,Z 203.679,A -85,B 0,C 180,E1 -15437.016,E2 -15437.016} C_VEL
LIN {X 0,Y 319.539,Z 203.68,A -85,B 0,C 180,E1 -15440.369,E2 -15440.369} C_VEL
LIN {X 0,Y 319.552,Z 203.679,A -85,B 0,C 180,E1 -15444.016,E2 -15444.016} C_VEL
LIN {X 0,Y 319.57,Z 203.672,A -85,B 0,C 180,E1 -15446.685,E2 -15446.685} C_VEL
LIN {X 0,Y 319.577,Z 203.674,A -85,B 0,C 180,E1 -15449.474,E2 -15449.474} C_VEL
LIN {X 0,Y 318.961,Z 203.753,A -85,B 0,C 180,E1 -15450.526,E2 -15450.526} C_VEL
LIN {X 0,Y 316.151,Z 204.104,A -85,B 0,C 180,E1 -15452.238,E2 -15452.238} C_VEL
LIN {X 0,Y 313.723,Z 204.406,A -85,B 0,C 180,E1 -15453.626,E2 -15453.626} C_VEL
LIN {X 0,Y 312.65,Z 204.53,A -85,B 0,C 180,E1 -15454.7,E2 -15454.7} C_VEL
LIN {X 0,Y 312.547,Z 204.541,A -85,B 0,C 180,E1 -15455.064,E2 -15455.064} C_VEL
LIN {X 0,Y 312.544,Z 204.547,A -85,B 0,C 180,E1 -15458.913,E2 -15458.913} C_VEL
LIN {X 0,Y 312.628,Z 204.541,A -85,B 0,C 180,E1 -15461.656,E2 -15461.656} C_VEL
LIN {X 0,Y 312.683,Z 204.527,A -85,B 0,C 180,E1 -15465.686,E2 -15465.686} C_VEL
LIN {X 0,Y 312.688,Z 204.523,A -85,B 0,C 180,E1 -15469.641,E2 -15469.641} C_VEL
LIN {X 0,Y 312.842,Z 204.514,A -85,B 0,C 180,E1 -15472.253,E2 -15472.253} C_VEL
LIN {X 0,Y 312.704,Z 204.522,A -85,B 0,C 180,E1 -15474.842,E2 -15474.842} C_VEL
LIN {X 0,Y 312.979,Z 204.495,A -85,B 0,C 180,E1 -15478.713,E2 -15478.713} C_VEL
LIN {X 0,Y 312.979,Z 204.494,A -85,B 0,C 180,E1 -15481.287,E2 -15481.287} C_VEL
LIN {X 0,Y 312.702,Z 204.525,A -85,B 0,C 180,E1 -15485.158,E2 -15485.158} C_VEL
LIN {X 0,Y 312.861,Z 204.512,A -85,B 0,C 180,E1 -15487.746,E2 -15487.746} C_VEL
LIN {X 0,Y 312.658,Z 204.539,A -85,B 0,C 180,E1 -15491.672,E2 -15491.672} C_VEL
LIN {X 0,Y 312.657,Z 204.54,A -85,B 0,C 180,E1 -15494.866,E2 -15494.866} C_VEL
LIN {X 0,Y 312.537,Z 204.555,A -85,B 0,C 180,E1 -15499.194,E2 -15499.194} C_VEL
LIN {X 0,Y 312.507,Z 204.559,A -85,B 0,C 180,E1 -15502.777,E2 -15502.777} C_VEL
LIN {X 0,Y 312.472,Z 204.564,A -85,B 0,C 180,E1 -15506.733,E2 -15506.733} C_VEL
LIN {X 0,Y 312.485,Z 204.563,A -85,B 0,C 180,E1 -15509.656,E2 -15509.656} C_VEL
LIN {X 0,Y 312.51,Z 204.555,A -85,B 0,C 180,E1 -15513.69,E2 -15513.69} C_VEL
LIN {X 0,Y 312.505,Z 204.557,A -85,B 0,C 180,E1 -15517.388,E2 -15517.388} C_VEL
LIN {X 0,Y 312.432,Z 204.55,A -85,B 0,C 180,E1 -15520.718,E2 -15520.718} C_VEL
LIN {X 0,Y 312.507,Z 204.67,A -85,B 0,C 180,E1 -15522.86,E2 -15522.86} C_VEL
LIN {X 0,Y 314.413,Z 212.555,A -85,B 0,C 180,E1 -15526.636,E2 -15526.636} C_VEL
LIN {X 0,Y 316.43,Z 221.045,A -85,B 0,C 180,E1 -15530.291,E2 -15530.291} C_VEL
LIN {X 0,Y 318.581,Z 230.714,A -85,B 0,C 180,E1 -15534.116,E2 -15534.116} C_VEL
LIN {X 0,Y 320.002,Z 237.762,A -85,B 0,C 180,E1 -15536.7,E2 -15536.7} C_VEL
LIN {X 0,Y 319.73,Z 241.038,A -85,B 0,C 180,E1 -15537.791,E2 -15537.791} C_VEL
LIN {X 0,Y 316.927,Z 253.978,A -85,B 0,C 180,E1 -15541.888,E2 -15541.888} C_VEL
LIN {X 0,Y 314.679,Z 266.68,A -85,B 0,C 180,E1 -15545.948,E2 -15545.948} C_VEL
LIN {X 0,Y 313.378,Z 275.565,A -85,B 0,C 180,E1 -15548.845,E2 -15548.845} C_VEL
LIN {X 0,Y 314.4,Z 287.865,A -85,B 0,C 180,E1 -15549.423,E2 -15549.423} C_VEL
LIN {X 0,Y 314.932,Z 299.551,A -85,B 0,C 180,E1 -15550.201,E2 -15550.201} C_VEL
LIN {X 0,Y 315.493,Z 312.145,A -85,B 0,C 180,E1 -15551.326,E2 -15551.326} C_VEL
LIN {X 0,Y 315.444,Z 320.654,A -85,B 0,C 180,E1 -15552.163,E2 -15552.163} C_VEL
LIN {X 0,Y 314.348,Z 333.208,A -85,B 0,C 180,E1 -15553.44,E2 -15553.44} C_VEL
LIN {X 0,Y 313.503,Z 343.475,A -85,B 0,C 180,E1 -15554.753,E2 -15554.753} C_VEL
LIN {X 0,Y 312.639,Z 353.648,A -85,B 0,C 180,E1 -15556.349,E2 -15556.349} C_VEL
LIN {X 0,Y 312.025,Z 362.186,A -85,B 0,C 180,E1 -15557.976,E2 -15557.976} C_VEL
LIN {X 0,Y 311.452,Z 370.509,A -85,B 0,C 180,E1 -15559.93,E2 -15559.93} C_VEL
LIN {X 0,Y 311.243,Z 376.191,A -85,B 0,C 180,E1 -15561.562,E2 -15561.562} C_VEL
LIN {X 0,Y 311.112,Z 382.129,A -85,B 0,C 180,E1 -15563.7,E2 -15563.7} C_VEL
LIN {X 0,Y 311.081,Z 385.914,A -85,B 0,C 180,E1 -15565.466,E2 -15565.466} C_VEL
LIN {X 0,Y 311.175,Z 389.018,A -85,B 0,C 180,E1 -15567.413,E2 -15567.413} C_VEL
LIN {X 0,Y 311.211,Z 390.506,A -85,B 0,C 180,E1 -15568.708,E2 -15568.708} C_VEL
LIN {X 0,Y 311.209,Z 391.528,A -85,B 0,C 180,E1 -15570.002,E2 -15570.002} C_VEL
LIN {X 0,Y 311.163,Z 392.088,A -85,B 0,C 180,E1 -15571.296,E2 -15571.296} C_VEL
LIN {X 0,Y 310.917,Z 391.97,A -85,B 0,C 180,E1 -15573.89,E2 -15573.89} C_VEL
LIN {X 0,Y 310.874,Z 390.725,A -85,B 0,C 180,E1 -15575.89,E2 -15575.89} C_VEL
LIN {X 0,Y 311.06,Z 388.639,A -85,B 0,C 180,E1 -15577.793,E2 -15577.793} C_VEL
LIN {X 0,Y 311.516,Z 385.582,A -85,B 0,C 180,E1 -15579.743,E2 -15579.743} C_VEL
LIN {X 0,Y 312.29,Z 381.547,A -85,B 0,C 180,E1 -15581.687,E2 -15581.687} C_VEL
LIN {X 0,Y 313.446,Z 376.449,A -85,B 0,C 180,E1 -15583.618,E2 -15583.618} C_VEL
LIN {X 0,Y 315.048,Z 370.211,A -85,B 0,C 180,E1 -15585.529,E2 -15585.529} C_VEL
LIN {X 0,Y 316.708,Z 362.833,A -85,B 0,C 180,E1 -15587.406,E2 -15587.406} C_VEL
LIN {X 0,Y 319.224,Z 353.617,A -85,B 0,C 180,E1 -15589.285,E2 -15589.285} C_VEL
LIN {X 0,Y 322.126,Z 342.63,A -85,B 0,C 180,E1 -15591.101,E2 -15591.101} C_VEL
LIN {X 0,Y 324.887,Z 331.522,A -85,B 0,C 180,E1 -15592.581,E2 -15592.581} C_VEL
LIN {X 0,Y 326.978,Z 319.824,A -85,B 0,C 180,E1 -15593.936,E2 -15593.936} C_VEL
LIN {X 0,Y 328.008,Z 307.877,A -85,B 0,C 180,E1 -15595.205,E2 -15595.205} C_VEL
LIN {X 0,Y 327.741,Z 295.2,A -85,B 0,C 180,E1 -15596.528,E2 -15596.528} C_VEL
LIN {X 0,Y 326.39,Z 283.77,A -85,B 0,C 180,E1 -15597.758,E2 -15597.758} C_VEL
LIN {X 0,Y 324.163,Z 271.59,A -85,B 0,C 180,E1 -15599.224,E2 -15599.224} C_VEL
LIN {X 0,Y 325.277,Z 262.774,A -85,B 0,C 180,E1 -15601.236,E2 -15601.236} C_VEL
LIN {X 0,Y 327.077,Z 254.084,A -85,B 0,C 180,E1 -15603.595,E2 -15603.595} C_VEL
LIN {X 0,Y 327.369,Z 251.222,A -85,B 0,C 180,E1 -15604.671,E2 -15604.671} C_VEL
LIN {X 0,Y 327.263,Z 246.915,A -85,B 0,C 180,E1 -15606.965,E2 -15606.965} C_VEL
LIN {X 0,Y 327.328,Z 243.706,A -85,B 0,C 180,E1 -15609.38,E2 -15609.38} C_VEL
LIN {X 0,Y 326.925,Z 242.24,A -85,B 0,C 180,E1 -15611.793,E2 -15611.793} C_VEL
LIN {X 0,Y 326.446,Z 242,A -85,B 0,C 180,E1 -15613.547,E2 -15613.547} C_VEL
LIN {X 0,Y 325.78,Z 242.59,A -85,B 0,C 180,E1 -15616.343,E2 -15616.343} C_VEL
LIN {X 0,Y 325.246,Z 244.453,A -85,B 0,C 180,E1 -15619.59,E2 -15619.59} C_VEL
LIN {X 0,Y 324.994,Z 245.794,A -85,B 0,C 180,E1 -15621.162,E2 -15621.162} C_VEL
LIN {X 0,Y 324.324,Z 248.188,A -85,B 0,C 180,E1 -15623.302,E2 -15623.302} C_VEL
LIN {X 0,Y 321.425,Z 255.895,A -85,B 0,C 180,E1 -15628.348,E2 -15628.348} C_VEL
LIN {X 0,Y 320.632,Z 259.155,A -85,B 0,C 180,E1 -15630.204,E2 -15630.204} C_VEL
LIN {X 0,Y 325.62,Z 271.599,A -85,B 0,C 180,E1 -15632.589,E2 -15632.589} C_VEL
LIN {X 0,Y 328.746,Z 282.656,A -85,B 0,C 180,E1 -15634.44,E2 -15634.44} C_VEL
LIN {X 0,Y 330.354,Z 291.815,A -85,B 0,C 180,E1 -15635.879,E2 -15635.879} C_VEL
LIN {X 0,Y 330.557,Z 293.71,A -85,B 0,C 180,E1 -15636.174,E2 -15636.174} C_VEL
LIN {X 0,Y 328.11,Z 305.223,A -85,B 0,C 180,E1 -15637.492,E2 -15637.492} C_VEL
LIN {X 0,Y 325.231,Z 316.671,A -85,B 0,C 180,E1 -15639.111,E2 -15639.111} C_VEL
LIN {X 0,Y 322.448,Z 326.842,A -85,B 0,C 180,E1 -15640.917,E2 -15640.917} C_VEL
LIN {X 0,Y 319.926,Z 335.217,A -85,B 0,C 180,E1 -15642.749,E2 -15642.749} C_VEL
LIN {X 0,Y 317.829,Z 342.074,A -85,B 0,C 180,E1 -15644.612,E2 -15644.612} C_VEL
LIN {X 0,Y 316.132,Z 347.628,A -85,B 0,C 180,E1 -15646.501,E2 -15646.501} C_VEL
LIN {X 0,Y 314.642,Z 352.084,A -85,B 0,C 180,E1 -15648.403,E2 -15648.403} C_VEL
LIN {X 0,Y 313.239,Z 356.264,A -85,B 0,C 180,E1 -15650.832,E2 -15650.832} C_VEL
LIN {X 0,Y 312.402,Z 358.007,A -85,B 0,C 180,E1 -15652.243,E2 -15652.243} C_VEL
LIN {X 0,Y 311.837,Z 359.853,A -85,B 0,C 180,E1 -15654.828,E2 -15654.828} C_VEL
LIN {X 0,Y 311.538,Z 360.211,A -85,B 0,C 180,E1 -15656.119,E2 -15656.119} C_VEL
LIN {X 0,Y 311.064,Z 359.667,A -85,B 0,C 180,E1 -15658.705,E2 -15658.705} C_VEL
LIN {X 0,Y 310.937,Z 358.807,A -85,B 0,C 180,E1 -15660,E2 -15660} C_VEL
LIN {X 0,Y 310.902,Z 357.519,A -85,B 0,C 180,E1 -15661.295,E2 -15661.295} C_VEL
LIN {X 0,Y 310.969,Z 354.783,A -85,B 0,C 180,E1 -15663.239,E2 -15663.239} C_VEL
LIN {X 0,Y 311.118,Z 351.023,A -85,B 0,C 180,E1 -15665.184,E2 -15665.184} C_VEL
LIN {X 0,Y 311.407,Z 345.259,A -85,B 0,C 180,E1 -15667.435,E2 -15667.435} C_VEL
LIN {X 0,Y 311.88,Z 338.852,A -85,B 0,C 180,E1 -15669.403,E2 -15669.403} C_VEL
LIN {X 0,Y 312.52,Z 330.98,A -85,B 0,C 180,E1 -15671.348,E2 -15671.348} C_VEL
LIN {X 0,Y 313.362,Z 321.283,A -85,B 0,C 180,E1 -15673.29,E2 -15673.29} C_VEL
LIN {X 0,Y 314.235,Z 311.38,A -85,B 0,C 180,E1 -15674.904,E2 -15674.904} C_VEL
LIN {X 0,Y 315.061,Z 301.198,A -85,B 0,C 180,E1 -15676.27,E2 -15676.27} C_VEL
LIN {X 0,Y 316.11,Z 288.634,A -85,B 0,C 180,E1 -15677.633,E2 -15677.633} C_VEL
LIN {X 0,Y 316.734,Z 277.418,A -85,B 0,C 180,E1 -15678.601,E2 -15678.601} C_VEL
LIN {X 0,Y 314.638,Z 264.23,A -85,B 0,C 180,E1 -15679.576,E2 -15679.576} C_VEL
LIN {X 0,Y 312.637,Z 250.975,A -85,B 0,C 180,E1 -15680.32,E2 -15680.32} C_VEL
LIN {X 0,Y 313.015,Z 242.975,A -85,B 0,C 180,E1 -15683.838,E2 -15683.838} C_VEL
LIN {X 0,Y 313.364,Z 235.018,A -85,B 0,C 180,E1 -15687.372,E2 -15687.372} C_VEL
LIN {X 0,Y 313.788,Z 226.866,A -85,B 0,C 180,E1 -15691.007,E2 -15691.007} C_VEL
LIN {X 0,Y 314.251,Z 218.481,A -85,B 0,C 180,E1 -15694.775,E2 -15694.775} C_VEL
LIN {X 0,Y 314.253,Z 214.981,A -85,B 0,C 180,E1 -15696.377,E2 -15696.377} C_VEL
LIN {X 0,Y 313.491,Z 209.621,A -85,B 0,C 180,E1 -15698.882,E2 -15698.882} C_VEL
LIN {X 0,Y 312.528,Z 204.557,A -85,B 0,C 180,E1 -15701.344,E2 -15701.344} C_VEL
LIN {X 0,Y 312.457,Z 204.565,A -85,B 0,C 180,E1 -15704.209,E2 -15704.209} C_VEL
LIN {X 0,Y 312.489,Z 204.562,A -85,B 0,C 180,E1 -15707.918,E2 -15707.918} C_VEL
LIN {X 0,Y 312.5,Z 204.56,A -85,B 0,C 180,E1 -15710.97,E2 -15710.97} C_VEL
LIN {X 0,Y 312.535,Z 204.559,A -85,B 0,C 180,E1 -15714.219,E2 -15714.219} C_VEL
LIN {X 0,Y 312.546,Z 204.659,A -85,B 0,C 180,E1 -15717.166,E2 -15717.166} C_VEL
LIN {X 0,Y 312.804,Z 206.375,A -85,B 0,C 180,E1 -15718.883,E2 -15718.883} C_VEL
LIN {X 0,Y 312.818,Z 209.494,A -85,B 0,C 180,E1 -15721.847,E2 -15721.847} C_VEL
LIN {X 0,Y 312.753,Z 212.648,A -85,B 0,C 180,E1 -15724.724,E2 -15724.724} C_VEL
LIN {X 0,Y 312.663,Z 215.874,A -85,B 0,C 180,E1 -15727.533,E2 -15727.533} C_VEL
LIN {X 0,Y 312.554,Z 220.851,A -85,B 0,C 180,E1 -15731.65,E2 -15731.65} C_VEL
LIN {X 0,Y 312.524,Z 224.168,A -85,B 0,C 180,E1 -15734.217,E2 -15734.217} C_VEL
LIN {X 0,Y 315.577,Z 234.917,A -85,B 0,C 180,E1 -15734.963,E2 -15734.963} C_VEL
LIN {X 0,Y 317.504,Z 243.625,A -85,B 0,C 180,E1 -15735.758,E2 -15735.758} C_VEL
LIN {X 0,Y 318.187,Z 247.847,A -85,B 0,C 180,E1 -15736.222,E2 -15736.222} C_VEL
LIN {X 0,Y 317.694,Z 255.165,A -85,B 0,C 180,E1 -15737.053,E2 -15737.053} C_VEL
LIN {X 0,Y 317.078,Z 261.864,A -85,B 0,C 180,E1 -15738.005,E2 -15738.005} C_VEL
LIN {X 0,Y 316.332,Z 268.132,A -85,B 0,C 180,E1 -15739.113,E2 -15739.113} C_VEL
LIN {X 0,Y 315.496,Z 273.884,A -85,B 0,C 180,E1 -15740.381,E2 -15740.381} C_VEL
LIN {X 0,Y 314.905,Z 278.408,A -85,B 0,C 180,E1 -15741.657,E2 -15741.657} C_VEL
LIN {X 0,Y 314.27,Z 282.021,A -85,B 0,C 180,E1 -15742.933,E2 -15742.933} C_VEL
LIN {X 0,Y 313.793,Z 285.974,A -85,B 0,C 180,E1 -15744.859,E2 -15744.859} C_VEL
LIN {X 0,Y 313.277,Z 287.845,A -85,B 0,C 180,E1 -15746.139,E2 -15746.139} C_VEL
LIN {X 0,Y 313.14,Z 289.112,A -85,B 0,C 180,E1 -15747.426,E2 -15747.426} C_VEL
LIN {X 0,Y 312.96,Z 289.88,A -85,B 0,C 180,E1 -15748.712,E2 -15748.712} C_VEL
LIN {X 0,Y 312.886,Z 290.147,A -85,B 0,C 180,E1 -15749.998,E2 -15749.998} C_VEL
LIN {X 0,Y 312.957,Z 289.917,A -85,B 0,C 180,E1 -15751.285,E2 -15751.285} C_VEL
LIN {X 0,Y 313.136,Z 289.2,A -85,B 0,C 180,E1 -15752.571,E2 -15752.571} C_VEL
LIN {X 0,Y 313.274,Z 287.987,A -85,B 0,C 180,E1 -15753.857,E2 -15753.857} C_VEL
LIN {X 0,Y 314.034,Z 285.039,A -85,B 0,C 180,E1 -15755.778,E2 -15755.778} C_VEL
LIN {X 0,Y 314.395,Z 280.667,A -85,B 0,C 180,E1 -15757.706,E2 -15757.706} C_VEL
LIN {X 0,Y 315.01,Z 277.741,A -85,B 0,C 180,E1 -15758.66,E2 -15758.66} C_VEL
LIN {X 0,Y 315.465,Z 274.344,A -85,B 0,C 180,E1 -15759.617,E2 -15759.617} C_VEL
LIN {X 0,Y 316.327,Z 268.721,A -85,B 0,C 180,E1 -15760.884,E2 -15760.884} C_VEL
LIN {X 0,Y 317.156,Z 261.602,A -85,B 0,C 180,E1 -15762.145,E2 -15762.145} C_VEL
LIN {X 0,Y 317.682,Z 254.695,A -85,B 0,C 180,E1 -15763.124,E2 -15763.124} C_VEL
LIN {X 0,Y 318.229,Z 247.89,A -85,B 0,C 180,E1 -15763.898,E2 -15763.898} C_VEL
LIN {X 0,Y 316.373,Z 238.033,A -85,B 0,C 180,E1 -15764.886,E2 -15764.886} C_VEL
LIN {X 0,Y 313.327,Z 226.837,A -85,B 0,C 180,E1 -15765.737,E2 -15765.737} C_VEL
LIN {X 0,Y 312.603,Z 224.147,A -85,B 0,C 180,E1 -15765.913,E2 -15765.913} C_VEL
LIN {X 0,Y 312.585,Z 219.324,A -85,B 0,C 180,E1 -15769.708,E2 -15769.708} C_VEL
LIN {X 0,Y 312.68,Z 215.568,A -85,B 0,C 180,E1 -15772.847,E2 -15772.847} C_VEL
LIN {X 0,Y 312.798,Z 211.227,A -85,B 0,C 180,E1 -15776.701,E2 -15776.701} C_VEL
LIN {X 0,Y 312.84,Z 208.121,A -85,B 0,C 180,E1 -15779.617,E2 -15779.617} C_VEL
LIN {X 0,Y 312.577,Z 204.971,A -85,B 0,C 180,E1 -15782.655,E2 -15782.655} C_VEL
LIN {X 0,Y 312.531,Z 204.557,A -85,B 0,C 180,E1 -15783.348,E2 -15783.348} C_VEL
LIN {X 0,Y 312.533,Z 204.557,A -85,B 0,C 180,E1 -15787.382,E2 -15787.382} C_VEL
LIN {X 0,Y 312.484,Z 204.562,A -85,B 0,C 180,E1 -15790.707,E2 -15790.707} C_VEL
LIN {X 0,Y 312.466,Z 204.56,A -85,B 0,C 180,E1 -15794.204,E2 -15794.204} C_VEL
LIN {X 0,Y 312.508,Z 204.558,A -85,B 0,C 180,E1 -15797.911,E2 -15797.911} C_VEL
LIN {X 0,Y 312.527,Z 204.554,A -85,B 0,C 180,E1 -15801.909,E2 -15801.909} C_VEL
LIN {X 0,Y 312.498,Z 204.555,A -85,B 0,C 180,E1 -15805.789,E2 -15805.789} C_VEL
LIN {X 0,Y 312.501,Z 204.551,A -85,B 0,C 180,E1 -15809.474,E2 -15809.474} C_VEL
LIN {X 0,Y 312.546,Z 204.552,A -85,B 0,C 180,E1 -15813.274,E2 -15813.274} C_VEL
LIN {X 0,Y 312.547,Z 204.541,A -85,B 0,C 180,E1 -15815.064,E2 -15815.064} C_VEL
LIN {X 0,Y 311.846,Z 204.637,A -85,B 0,C 180,E1 -15816.139,E2 -15816.139} C_VEL
LIN {X 0,Y 309.013,Z 204.993,A -85,B 0,C 180,E1 -15817.89,E2 -15817.89} C_VEL
LIN {X 0,Y 306.644,Z 205.284,A -85,B 0,C 180,E1 -15819.31,E2 -15819.31} C_VEL
LIN {X 0,Y 305.642,Z 205.406,A -85,B 0,C 180,E1 -15820.408,E2 -15820.408} C_VEL
LIN {X 0,Y 305.567,Z 205.416,A -85,B 0,C 180,E1 -15820.78,E2 -15820.78} C_VEL
LIN {X 0,Y 305.627,Z 205.401,A -85,B 0,C 180,E1 -15824.964,E2 -15824.964} C_VEL
LIN {X 0,Y 305.625,Z 205.404,A -85,B 0,C 180,E1 -15829.399,E2 -15829.399} C_VEL
LIN {X 0,Y 305.786,Z 205.393,A -85,B 0,C 180,E1 -15832.074,E2 -15832.074} C_VEL
LIN {X 0,Y 305.675,Z 205.398,A -85,B 0,C 180,E1 -15834.723,E2 -15834.723} C_VEL
LIN {X 0,Y 305.946,Z 205.371,A -85,B 0,C 180,E1 -15838.684,E2 -15838.684} C_VEL
LIN {X 0,Y 305.945,Z 205.371,A -85,B 0,C 180,E1 -15841.316,E2 -15841.316} C_VEL
LIN {X 0,Y 305.84,Z 205.388,A -85,B 0,C 180,E1 -15846.598,E2 -15846.598} C_VEL
LIN {X 0,Y 305.725,Z 205.393,A -85,B 0,C 180,E1 -15849.26,E2 -15849.26} C_VEL
LIN {X 0,Y 305.575,Z 205.412,A -85,B 0,C 180,E1 -15853.297,E2 -15853.297} C_VEL
LIN {X 0,Y 305.542,Z 205.427,A -85,B 0,C 180,E1 -15856.023,E2 -15856.023} C_VEL
LIN {X 0,Y 305.472,Z 205.436,A -85,B 0,C 180,E1 -15860.188,E2 -15860.188} C_VEL
LIN {X 0,Y 305.445,Z 205.44,A -85,B 0,C 180,E1 -15864.467,E2 -15864.467} C_VEL
LIN {X 0,Y 305.438,Z 205.441,A -85,B 0,C 180,E1 -15867.399,E2 -15867.399} C_VEL
LIN {X 0,Y 305.42,Z 205.441,A -85,B 0,C 180,E1 -15870.414,E2 -15870.414} C_VEL
LIN {X 0,Y 305.455,Z 205.431,A -85,B 0,C 180,E1 -15874.08,E2 -15874.08} C_VEL
LIN {X 0,Y 305.445,Z 205.436,A -85,B 0,C 180,E1 -15876.744,E2 -15876.744} C_VEL
LIN {X 0,Y 305.4,Z 205.426,A -85,B 0,C 180,E1 -15880.591,E2 -15880.591} C_VEL
LIN {X 0,Y 305.426,Z 205.589,A -85,B 0,C 180,E1 -15882.013,E2 -15882.013} C_VEL
LIN {X 0,Y 307.374,Z 213.511,A -85,B 0,C 180,E1 -15885.987,E2 -15885.987} C_VEL
LIN {X 0,Y 309.282,Z 221.49,A -85,B 0,C 180,E1 -15889.573,E2 -15889.573} C_VEL
LIN {X 0,Y 311.523,Z 231.557,A -85,B 0,C 180,E1 -15893.689,E2 -15893.689} C_VEL
LIN {X 0,Y 312.894,Z 238.149,A -85,B 0,C 180,E1 -15896.209,E2 -15896.209} C_VEL
LIN {X 0,Y 313.109,Z 239.828,A -85,B 0,C 180,E1 -15896.823,E2 -15896.823} C_VEL
LIN {X 0,Y 312.198,Z 244.737,A -85,B 0,C 180,E1 -15898.442,E2 -15898.442} C_VEL
LIN {X 0,Y 309.03,Z 259.636,A -85,B 0,C 180,E1 -15903.313,E2 -15903.313} C_VEL
LIN {X 0,Y 306.553,Z 274.092,A -85,B 0,C 180,E1 -15908.129,E2 -15908.129} C_VEL
LIN {X 0,Y 306.467,Z 274.848,A -85,B 0,C 180,E1 -15908.388,E2 -15908.388} C_VEL
LIN {X 0,Y 307.584,Z 287.758,A -85,B 0,C 180,E1 -15909.041,E2 -15909.041} C_VEL
LIN {X 0,Y 308.051,Z 299.723,A -85,B 0,C 180,E1 -15909.873,E2 -15909.873} C_VEL
LIN {X 0,Y 308.482,Z 310.773,A -85,B 0,C 180,E1 -15910.885,E2 -15910.885} C_VEL
LIN {X 0,Y 308.458,Z 320.03,A -85,B 0,C 180,E1 -15911.916,E2 -15911.916} C_VEL
LIN {X 0,Y 307.178,Z 334.874,A -85,B 0,C 180,E1 -15913.555,E2 -15913.555} C_VEL
LIN {X 0,Y 306.124,Z 346.259,A -85,B 0,C 180,E1 -15915.125,E2 -15915.125} C_VEL
LIN {X 0,Y 305.389,Z 355.505,A -85,B 0,C 180,E1 -15916.697,E2 -15916.697} C_VEL
LIN {X 0,Y 304.662,Z 365.053,A -85,B 0,C 180,E1 -15918.694,E2 -15918.694} C_VEL
LIN {X 0,Y 304.286,Z 372.746,A -85,B 0,C 180,E1 -15920.698,E2 -15920.698} C_VEL
LIN {X 0,Y 304.082,Z 378.864,A -85,B 0,C 180,E1 -15922.699,E2 -15922.699} C_VEL
LIN {X 0,Y 304.065,Z 383.665,A -85,B 0,C 180,E1 -15924.697,E2 -15924.697} C_VEL
LIN {X 0,Y 304.027,Z 387.26,A -85,B 0,C 180,E1 -15926.689,E2 -15926.689} C_VEL
LIN {X 0,Y 304.153,Z 389.781,A -85,B 0,C 180,E1 -15928.678,E2 -15928.678} C_VEL
LIN {X 0,Y 304.149,Z 390.898,A -85,B 0,C 180,E1 -15930.002,E2 -15930.002} C_VEL
LIN {X 0,Y 304.096,Z 391.559,A -85,B 0,C 180,E1 -15931.326,E2 -15931.326} C_VEL
LIN {X 0,Y 303.839,Z 391.76,A -85,B 0,C 180,E1 -15932.653,E2 -15932.653} C_VEL
LIN {X 0,Y 303.84,Z 391.572,A -85,B 0,C 180,E1 -15933.981,E2 -15933.981} C_VEL
LIN {X 0,Y 303.789,Z 390.6,A -85,B 0,C 180,E1 -15935.854,E2 -15935.854} C_VEL
LIN {X 0,Y 304.011,Z 388.527,A -85,B 0,C 180,E1 -15937.975,E2 -15937.975} C_VEL
LIN {X 0,Y 304.713,Z 384.47,A -85,B 0,C 180,E1 -15940.634,E2 -15940.634} C_VEL
LIN {X 0,Y 305.659,Z 380.276,A -85,B 0,C 180,E1 -15942.619,E2 -15942.619} C_VEL
LIN {X 0,Y 307.42,Z 374.023,A -85,B 0,C 180,E1 -15944.905,E2 -15944.905} C_VEL
LIN {X 0,Y 309.388,Z 366.209,A -85,B 0,C 180,E1 -15947.177,E2 -15947.177} C_VEL
LIN {X 0,Y 311.708,Z 358.045,A -85,B 0,C 180,E1 -15949.084,E2 -15949.084} C_VEL
LIN {X 0,Y 314.615,Z 348.151,A -85,B 0,C 180,E1 -15950.943,E2 -15950.943} C_VEL
LIN {X 0,Y 317.658,Z 337.291,A -85,B 0,C 180,E1 -15952.609,E2 -15952.609} C_VEL
LIN {X 0,Y 320.186,Z 326.711,A -85,B 0,C 180,E1 -15953.96,E2 -15953.96} C_VEL
LIN {X 0,Y 322.056,Z 314.266,A -85,B 0,C 180,E1 -15955.4,E2 -15955.4} C_VEL
LIN {X 0,Y 322.582,Z 302.495,A -85,B 0,C 180,E1 -15956.714,E2 -15956.714} C_VEL
LIN {X 0,Y 322.115,Z 291.856,A -85,B 0,C 180,E1 -15957.908,E2 -15957.908} C_VEL
LIN {X 0,Y 320.164,Z 278.171,A -85,B 0,C 180,E1 -15959.556,E2 -15959.556} C_VEL
LIN {X 0,Y 318.935,Z 271.043,A -85,B 0,C 180,E1 -15960.537,E2 -15960.537} C_VEL
LIN {X 0,Y 320.474,Z 261.883,A -85,B 0,C 180,E1 -15962.853,E2 -15962.853} C_VEL
LIN {X 0,Y 321.601,Z 257.32,A -85,B 0,C 180,E1 -15964.179,E2 -15964.179} C_VEL
LIN {X 0,Y 321.801,Z 254.362,A -85,B 0,C 180,E1 -15965.41,E2 -15965.41} C_VEL
LIN {X 0,Y 321.691,Z 250.316,A -85,B 0,C 180,E1 -15967.715,E2 -15967.715} C_VEL
LIN {X 0,Y 321.721,Z 248.233,A -85,B 0,C 180,E1 -15969.311,E2 -15969.311} C_VEL
LIN {X 0,Y 321.46,Z 246.9,A -85,B 0,C 180,E1 -15970.988,E2 -15970.988} C_VEL
LIN {X 0,Y 320.955,Z 246.282,A -85,B 0,C 180,E1 -15972.752,E2 -15972.752} C_VEL
LIN {X 0,Y 320.176,Z 246.376,A -85,B 0,C 180,E1 -15975.379,E2 -15975.379} C_VEL
LIN {X 0,Y 319.416,Z 247.759,A -85,B 0,C 180,E1 -15978.694,E2 -15978.694} C_VEL
LIN {X 0,Y 319.061,Z 248.995,A -85,B 0,C 180,E1 -15980.441,E2 -15980.441} C_VEL
LIN {X 0,Y 318.414,Z 251.091,A -85,B 0,C 180,E1 -15982.618,E2 -15982.618} C_VEL
LIN {X 0,Y 316.804,Z 254.566,A -85,B 0,C 180,E1 -15985.168,E2 -15985.168} C_VEL
LIN {X 0,Y 314.922,Z 259.903,A -85,B 0,C 180,E1 -15988.647,E2 -15988.647} C_VEL
LIN {X 0,Y 319.609,Z 271.94,A -85,B 0,C 180,E1 -15991.245,E2 -15991.245} C_VEL
LIN {X 0,Y 322.012,Z 279.715,A -85,B 0,C 180,E1 -15992.72,E2 -15992.72} C_VEL
LIN {X 0,Y 324.183,Z 289.923,A -85,B 0,C 180,E1 -15994.503,E2 -15994.503} C_VEL
LIN {X 0,Y 324.899,Z 295.755,A -85,B 0,C 180,E1 -15995.466,E2 -15995.466} C_VEL
LIN {X 0,Y 322.251,Z 307.38,A -85,B 0,C 180,E1 -15996.886,E2 -15996.886} C_VEL
LIN {X 0,Y 319.475,Z 317.566,A -85,B 0,C 180,E1 -15998.378,E2 -15998.378} C_VEL
LIN {X 0,Y 316.505,Z 327.589,A -85,B 0,C 180,E1 -16000.207,E2 -16000.207} C_VEL
LIN {X 0,Y 313.773,Z 335.887,A -85,B 0,C 180,E1 -16002.063,E2 -16002.063} C_VEL
LIN {X 0,Y 311.162,Z 343.655,A -85,B 0,C 180,E1 -16004.274,E2 -16004.274} C_VEL
LIN {X 0,Y 309.374,Z 348.982,A -85,B 0,C 180,E1 -16006.2,E2 -16006.2} C_VEL
LIN {X 0,Y 307.793,Z 353.234,A -85,B 0,C 180,E1 -16008.141,E2 -16008.141} C_VEL
LIN {X 0,Y 306.316,Z 357.178,A -85,B 0,C 180,E1 -16010.608,E2 -16010.608} C_VEL
LIN {X 0,Y 305.424,Z 358.8,A -85,B 0,C 180,E1 -16012.064,E2 -16012.064} C_VEL
LIN {X 0,Y 304.975,Z 359.836,A -85,B 0,C 180,E1 -16013.384,E2 -16013.384} C_VEL
LIN {X 0,Y 304.777,Z 360.467,A -85,B 0,C 180,E1 -16014.708,E2 -16014.708} C_VEL
LIN {X 0,Y 304.468,Z 360.692,A -85,B 0,C 180,E1 -16016.029,E2 -16016.029} C_VEL
LIN {X 0,Y 303.973,Z 359.986,A -85,B 0,C 180,E1 -16018.675,E2 -16018.675} C_VEL
LIN {X 0,Y 303.84,Z 359.02,A -85,B 0,C 180,E1 -16020,E2 -16020} C_VEL
LIN {X 0,Y 303.809,Z 357.62,A -85,B 0,C 180,E1 -16021.326,E2 -16021.326} C_VEL
LIN {X 0,Y 303.897,Z 354.739,A -85,B 0,C 180,E1 -16023.315,E2 -16023.315} C_VEL
LIN {X 0,Y 304.027,Z 350.829,A -85,B 0,C 180,E1 -16025.306,E2 -16025.306} C_VEL
LIN {X 0,Y 304.317,Z 345.244,A -85,B 0,C 180,E1 -16027.48,E2 -16027.48} C_VEL
LIN {X 0,Y 304.843,Z 338.284,A -85,B 0,C 180,E1 -16029.622,E2 -16029.622} C_VEL
LIN {X 0,Y 305.523,Z 330.196,A -85,B 0,C 180,E1 -16031.612,E2 -16031.612} C_VEL
LIN {X 0,Y 306.228,Z 322.037,A -85,B 0,C 180,E1 -16033.268,E2 -16033.268} C_VEL
LIN {X 0,Y 307.174,Z 312.241,A -85,B 0,C 180,E1 -16034.916,E2 -16034.916} C_VEL
LIN {X 0,Y 308.037,Z 301,A -85,B 0,C 180,E1 -16036.461,E2 -16036.461} C_VEL
LIN {X 0,Y 309.04,Z 289.828,A -85,B 0,C 180,E1 -16037.708,E2 -16037.708} C_VEL
LIN {X 0,Y 309.765,Z 279.226,A -85,B 0,C 180,E1 -16038.666,E2 -16038.666} C_VEL
LIN {X 0,Y 308.123,Z 267.863,A -85,B 0,C 180,E1 -16039.556,E2 -16039.556} C_VEL
LIN {X 0,Y 305.96,Z 254.038,A -85,B 0,C 180,E1 -16040.396,E2 -16040.396} C_VEL
LIN {X 0,Y 305.625,Z 251.356,A -85,B 0,C 180,E1 -16040.529,E2 -16040.529} C_VEL
LIN {X 0,Y 306.046,Z 242.619,A -85,B 0,C 180,E1 -16044.416,E2 -16044.416} C_VEL
LIN {X 0,Y 306.393,Z 234.537,A -85,B 0,C 180,E1 -16048.049,E2 -16048.049} C_VEL
LIN {X 0,Y 306.929,Z 225.608,A -85,B 0,C 180,E1 -16052.087,E2 -16052.087} C_VEL
LIN {X 0,Y 307.29,Z 217.732,A -85,B 0,C 180,E1 -16055.677,E2 -16055.677} C_VEL
LIN {X 0,Y 306.794,Z 212.352,A -85,B 0,C 180,E1 -16058.208,E2 -16058.208} C_VEL
LIN {X 0,Y 305.465,Z 205.437,A -85,B 0,C 180,E1 -16061.617,E2 -16061.617} C_VEL
LIN {X 0,Y 305.406,Z 205.44,A -85,B 0,C 180,E1 -16065.51,E2 -16065.51} C_VEL
LIN {X 0,Y 305.446,Z 205.439,A -85,B 0,C 180,E1 -16068.142,E2 -16068.142} C_VEL
LIN {X 0,Y 305.467,Z 205.438,A -85,B 0,C 180,E1 -16071.594,E2 -16071.594} C_VEL
LIN {X 0,Y 305.466,Z 205.439,A -85,B 0,C 180,E1 -16074.886,E2 -16074.886} C_VEL
LIN {X 0,Y 305.51,Z 205.566,A -85,B 0,C 180,E1 -16076.685,E2 -16076.685} C_VEL
LIN {X 0,Y 305.817,Z 208.494,A -85,B 0,C 180,E1 -16079.628,E2 -16079.628} C_VEL
LIN {X 0,Y 305.801,Z 211.691,A -85,B 0,C 180,E1 -16082.634,E2 -16082.634} C_VEL
LIN {X 0,Y 305.701,Z 214.869,A -85,B 0,C 180,E1 -16085.554,E2 -16085.554} C_VEL
LIN {X 0,Y 305.609,Z 218.165,A -85,B 0,C 180,E1 -16088.409,E2 -16088.409} C_VEL
LIN {X 0,Y 305.584,Z 221.546,A -85,B 0,C 180,E1 -16091.216,E2 -16091.216} C_VEL
LIN {X 0,Y 305.53,Z 224.903,A -85,B 0,C 180,E1 -16093.782,E2 -16093.782} C_VEL
LIN {X 0,Y 308.42,Z 234.847,A -85,B 0,C 180,E1 -16094.486,E2 -16094.486} C_VEL
LIN {X 0,Y 310.449,Z 243.569,A -85,B 0,C 180,E1 -16095.293,E2 -16095.293} C_VEL
LIN {X 0,Y 311.403,Z 249.052,A -85,B 0,C 180,E1 -16095.909,E2 -16095.909} C_VEL
LIN {X 0,Y 310.883,Z 256.125,A -85,B 0,C 180,E1 -16096.735,E2 -16096.735} C_VEL
LIN {X 0,Y 310.118,Z 263.989,A -85,B 0,C 180,E1 -16097.898,E2 -16097.898} C_VEL
LIN {X 0,Y 308.985,Z 272.234,A -85,B 0,C 180,E1 -16099.514,E2 -16099.514} C_VEL
LIN {X 0,Y 308.184,Z 277.299,A -85,B 0,C 180,E1 -16100.813,E2 -16100.813} C_VEL
LIN {X 0,Y 307.465,Z 281.34,A -85,B 0,C 180,E1 -16102.116,E2 -16102.116} C_VEL
LIN {X 0,Y 307.053,Z 285.795,A -85,B 0,C 180,E1 -16104.086,E2 -16104.086} C_VEL
LIN {X 0,Y 306.267,Z 288.821,A -85,B 0,C 180,E1 -16106.051,E2 -16106.051} C_VEL
LIN {X 0,Y 306.121,Z 290.086,A -85,B 0,C 180,E1 -16107.367,E2 -16107.367} C_VEL
LIN {X 0,Y 305.935,Z 290.854,A -85,B 0,C 180,E1 -16108.682,E2 -16108.682} C_VEL
LIN {X 0,Y 305.859,Z 291.121,A -85,B 0,C 180,E1 -16109.998,E2 -16109.998} C_VEL
LIN {X 0,Y 305.932,Z 290.89,A -85,B 0,C 180,E1 -16111.315,E2 -16111.315} C_VEL
LIN {X 0,Y 306.117,Z 290.174,A -85,B 0,C 180,E1 -16112.63,E2 -16112.63} C_VEL
LIN {X 0,Y 306.264,Z 288.962,A -85,B 0,C 180,E1 -16113.946,E2 -16113.946} C_VEL
LIN {X 0,Y 307.044,Z 286.02,A -85,B 0,C 180,E1 -16115.91,E2 -16115.91} C_VEL
LIN {X 0,Y 307.431,Z 281.658,A -85,B 0,C 180,E1 -16117.882,E2 -16117.882} C_VEL
LIN {X 0,Y 308.065,Z 278.742,A -85,B 0,C 180,E1 -16118.856,E2 -16118.856} C_VEL
LIN {X 0,Y 308.541,Z 275.362,A -85,B 0,C 180,E1 -16119.835,E2 -16119.835} C_VEL
LIN {X 0,Y 309.44,Z 269.778,A -85,B 0,C 180,E1 -16121.129,E2 -16121.129} C_VEL
LIN {X 0,Y 310.308,Z 262.67,A -85,B 0,C 180,E1 -16122.423,E2 -16122.423} C_VEL
LIN {X 0,Y 310.866,Z 255.704,A -85,B 0,C 180,E1 -16123.438,E2 -16123.438} C_VEL
LIN {X 0,Y 311.422,Z 249.131,A -85,B 0,C 180,E1 -16124.211,E2 -16124.211} C_VEL
LIN {X 0,Y 309.639,Z 239.577,A -85,B 0,C 180,E1 -16125.21,E2 -16125.21} C_VEL
LIN {X 0,Y 306.859,Z 229.206,A -85,B 0,C 180,E1 -16126.052,E2 -16126.052} C_VEL
LIN {X 0,Y 305.595,Z 224.762,A -85,B 0,C 180,E1 -16126.374,E2 -16126.374} C_VEL
LIN {X 0,Y 305.598,Z 220.004,A -85,B 0,C 180,E1 -16130.178,E2 -16130.178} C_VEL
LIN {X 0,Y 305.73,Z 215.046,A -85,B 0,C 180,E1 -16134.44,E2 -16134.44} C_VEL
LIN {X 0,Y 305.82,Z 211.822,A -85,B 0,C 180,E1 -16137.36,E2 -16137.36} C_VEL
LIN {X 0,Y 305.805,Z 208.63,A -85,B 0,C 180,E1 -16140.369,E2 -16140.369} C_VEL
LIN {X 0,Y 305.473,Z 205.436,A -85,B 0,C 180,E1 -16143.653,E2 -16143.653} C_VEL
LIN {X 0,Y 305.491,Z 205.432,A -85,B 0,C 180,E1 -16146.735,E2 -16146.735} C_VEL
LIN {X 0,Y 305.449,Z 205.438,A -85,B 0,C 180,E1 -16150.598,E2 -16150.598} C_VEL
LIN {X 0,Y 305.412,Z 205.439,A -85,B 0,C 180,E1 -16154.491,E2 -16154.491} C_VEL
LIN {X 0,Y 305.457,Z 205.436,A -85,B 0,C 180,E1 -16158.146,E2 -16158.146} C_VEL
LIN {X 0,Y 305.487,Z 205.431,A -85,B 0,C 180,E1 -16161.599,E2 -16161.599} C_VEL
LIN {X 0,Y 305.455,Z 205.436,A -85,B 0,C 180,E1 -16164.886,E2 -16164.886} C_VEL
LIN {X 0,Y 305.448,Z 205.439,A -85,B 0,C 180,E1 -16168.352,E2 -16168.352} C_VEL
LIN {X 0,Y 305.512,Z 205.423,A -85,B 0,C 180,E1 -16171.113,E2 -16171.113} C_VEL
LIN {X 0,Y 305.498,Z 205.419,A -85,B 0,C 180,E1 -16175.059,E2 -16175.059} C_VEL
LIN {X 0,Y 305.49,Z 205.427,A -85,B 0,C 180,E1 -16178.402,E2 -16178.402} C_VEL
LIN {X 0,Y 305.567,Z 205.416,A -85,B 0,C 180,E1 -16180.78,E2 -16180.78} C_VEL
LIN {X 0,Y 304.921,Z 205.504,A -85,B 0,C 180,E1 -16181.881,E2 -16181.881} C_VEL
LIN {X 0,Y 302.095,Z 205.856,A -85,B 0,C 180,E1 -16183.673,E2 -16183.673} C_VEL
LIN {X 0,Y 299.678,Z 206.156,A -85,B 0,C 180,E1 -16185.127,E2 -16185.127} C_VEL
LIN {X 0,Y 298.623,Z 206.285,A -85,B 0,C 180,E1 -16186.253,E2 -16186.253} C_VEL
LIN {X 0,Y 298.529,Z 206.295,A -85,B 0,C 180,E1 -16186.634,E2 -16186.634} C_VEL
LIN {X 0,Y 298.717,Z 206.267,A -85,B 0,C 180,E1 -16191.155,E2 -16191.155} C_VEL
LIN {X 0,Y 298.776,Z 206.266,A -85,B 0,C 180,E1 -16193.246,E2 -16193.246} C_VEL
LIN {X 0,Y 298.913,Z 206.247,A -85,B 0,C 180,E1 -16198.653,E2 -16198.653} C_VEL
LIN {X 0,Y 298.912,Z 206.247,A -85,B 0,C 180,E1 -16201.347,E2 -16201.347} C_VEL
LIN {X 0,Y 298.785,Z 206.268,A -85,B 0,C 180,E1 -16206.754,E2 -16206.754} C_VEL
LIN {X 0,Y 298.67,Z 206.272,A -85,B 0,C 180,E1 -16209.481,E2 -16209.481} C_VEL
LIN {X 0,Y 298.534,Z 206.289,A -85,B 0,C 180,E1 -16213.616,E2 -16213.616} C_VEL
LIN {X 0,Y 298.475,Z 206.303,A -85,B 0,C 180,E1 -16216.413,E2 -16216.413} C_VEL
LIN {X 0,Y 298.431,Z 206.313,A -85,B 0,C 180,E1 -16219.618,E2 -16219.618} C_VEL
LIN {X 0,Y 298.377,Z 206.321,A -85,B 0,C 180,E1 -16223.604,E2 -16223.604} C_VEL
LIN {X 0,Y 298.391,Z 206.318,A -85,B 0,C 180,E1 -16226.584,E2 -16226.584} C_VEL
LIN {X 0,Y 298.382,Z 206.319,A -85,B 0,C 180,E1 -16229.645,E2 -16229.645} C_VEL
LIN {X 0,Y 298.383,Z 206.317,A -85,B 0,C 180,E1 -16232.802,E2 -16232.802} C_VEL
LIN {X 0,Y 298.419,Z 206.311,A -85,B 0,C 180,E1 -16236.804,E2 -16236.804} C_VEL
LIN {X 0,Y 298.359,Z 206.303,A -85,B 0,C 180,E1 -16241.043,E2 -16241.043} C_VEL
LIN {X 0,Y 300.005,Z 213.143,A -85,B 0,C 180,E1 -16244.651,E2 -16244.651} C_VEL
LIN {X 0,Y 301.796,Z 220.527,A -85,B 0,C 180,E1 -16248.176,E2 -16248.176} C_VEL
LIN {X 0,Y 303.702,Z 229.083,A -85,B 0,C 180,E1 -16251.887,E2 -16251.887} C_VEL
LIN {X 0,Y 305.624,Z 237.921,A -85,B 0,C 180,E1 -16255.441,E2 -16255.441} C_VEL
LIN {X 0,Y 306.103,Z 241.996,A -85,B 0,C 180,E1 -16256.958,E2 -16256.958} C_VEL
LIN {X 0,Y 303.611,Z 252.598,A -85,B 0,C 180,E1 -16260.537,E2 -16260.537} C_VEL
LIN {X 0,Y 301.086,Z 265.129,A -85,B 0,C 180,E1 -16264.789,E2 -16264.789} C_VEL
LIN {X 0,Y 299.518,Z 274.275,A -85,B 0,C 180,E1 -16267.951,E2 -16267.951} C_VEL
LIN {X 0,Y 300.713,Z 287.344,A -85,B 0,C 180,E1 -16268.621,E2 -16268.621} C_VEL
LIN {X 0,Y 301.156,Z 299.676,A -85,B 0,C 180,E1 -16269.512,E2 -16269.512} C_VEL
LIN {X 0,Y 301.535,Z 311.149,A -85,B 0,C 180,E1 -16270.604,E2 -16270.604} C_VEL
LIN {X 0,Y 301.419,Z 321.504,A -85,B 0,C 180,E1 -16271.831,E2 -16271.831} C_VEL
LIN {X 0,Y 300.539,Z 329.457,A -85,B 0,C 180,E1 -16272.831,E2 -16272.831} C_VEL
LIN {X 0,Y 299.522,Z 341.333,A -85,B 0,C 180,E1 -16274.361,E2 -16274.361} C_VEL
LIN {X 0,Y 298.613,Z 351.779,A -85,B 0,C 180,E1 -16276.042,E2 -16276.042} C_VEL
LIN {X 0,Y 297.799,Z 362,A -85,B 0,C 180,E1 -16278.085,E2 -16278.085} C_VEL
LIN {X 0,Y 297.278,Z 370.147,A -85,B 0,C 180,E1 -16280.133,E2 -16280.133} C_VEL
LIN {X 0,Y 297.095,Z 375.724,A -85,B 0,C 180,E1 -16281.842,E2 -16281.842} C_VEL
LIN {X 0,Y 297.013,Z 381.708,A -85,B 0,C 180,E1 -16284.141,E2 -16284.141} C_VEL
LIN {X 0,Y 296.927,Z 385.255,A -85,B 0,C 180,E1 -16285.93,E2 -16285.93} C_VEL
LIN {X 0,Y 297.032,Z 387.408,A -85,B 0,C 180,E1 -16287.289,E2 -16287.289} C_VEL
LIN {X 0,Y 297.095,Z 389.041,A -85,B 0,C 180,E1 -16288.646,E2 -16288.646} C_VEL
LIN {X 0,Y 297.09,Z 390.223,A -85,B 0,C 180,E1 -16290.002,E2 -16290.002} C_VEL
LIN {X 0,Y 297.03,Z 390.981,A -85,B 0,C 180,E1 -16291.358,E2 -16291.358} C_VEL
LIN {X 0,Y 296.755,Z 391.291,A -85,B 0,C 180,E1 -16292.717,E2 -16292.717} C_VEL
LIN {X 0,Y 296.765,Z 391.176,A -85,B 0,C 180,E1 -16294.076,E2 -16294.076} C_VEL
LIN {X 0,Y 296.747,Z 389.745,A -85,B 0,C 180,E1 -16296.802,E2 -16296.802} C_VEL
LIN {X 0,Y 296.956,Z 388.437,A -85,B 0,C 180,E1 -16298.165,E2 -16298.165} C_VEL
LIN {X 0,Y 297.719,Z 384.557,A -85,B 0,C 180,E1 -16300.887,E2 -16300.887} C_VEL
LIN {X 0,Y 298.724,Z 380.555,A -85,B 0,C 180,E1 -16302.917,E2 -16302.917} C_VEL
LIN {X 0,Y 300.31,Z 375.509,A -85,B 0,C 180,E1 -16304.919,E2 -16304.919} C_VEL
LIN {X 0,Y 302.321,Z 368.27,A -85,B 0,C 180,E1 -16307.243,E2 -16307.243} C_VEL
LIN {X 0,Y 304.647,Z 360.659,A -85,B 0,C 180,E1 -16309.194,E2 -16309.194} C_VEL
LIN {X 0,Y 307.609,Z 351.498,A -85,B 0,C 180,E1 -16311.092,E2 -16311.092} C_VEL
LIN {X 0,Y 310.952,Z 340.5,A -85,B 0,C 180,E1 -16312.948,E2 -16312.948} C_VEL
LIN {X 0,Y 313.995,Z 329.48,A -85,B 0,C 180,E1 -16314.463,E2 -16314.463} C_VEL
LIN {X 0,Y 316.168,Z 318.133,A -85,B 0,C 180,E1 -16315.866,E2 -16315.866} C_VEL
LIN {X 0,Y 317.208,Z 306.655,A -85,B 0,C 180,E1 -16317.222,E2 -16317.222} C_VEL
LIN {X 0,Y 317.1,Z 294.71,A -85,B 0,C 180,E1 -16318.653,E2 -16318.653} C_VEL
LIN {X 0,Y 315.729,Z 281.916,A -85,B 0,C 180,E1 -16320.293,E2 -16320.293} C_VEL
LIN {X 0,Y 313.894,Z 270.691,A -85,B 0,C 180,E1 -16321.918,E2 -16321.918} C_VEL
LIN {X 0,Y 315.909,Z 261.636,A -85,B 0,C 180,E1 -16324.428,E2 -16324.428} C_VEL
LIN {X 0,Y 316.215,Z 259.367,A -85,B 0,C 180,E1 -16325.302,E2 -16325.302} C_VEL
LIN {X 0,Y 316.151,Z 256.269,A -85,B 0,C 180,E1 -16326.886,E2 -16326.886} C_VEL
LIN {X 0,Y 316.114,Z 253.252,A -85,B 0,C 180,E1 -16328.909,E2 -16328.909} C_VEL
LIN {X 0,Y 316.075,Z 251.876,A -85,B 0,C 180,E1 -16330.154,E2 -16330.154} C_VEL
LIN {X 0,Y 315.342,Z 250.577,A -85,B 0,C 180,E1 -16332.653,E2 -16332.653} C_VEL
LIN {X 0,Y 314.315,Z 250.584,A -85,B 0,C 180,E1 -16335.687,E2 -16335.687} C_VEL
LIN {X 0,Y 313.698,Z 251.295,A -85,B 0,C 180,E1 -16337.77,E2 -16337.77} C_VEL
LIN {X 0,Y 313.201,Z 252.38,A -85,B 0,C 180,E1 -16339.726,E2 -16339.726} C_VEL
LIN {X 0,Y 312.562,Z 254.155,A -85,B 0,C 180,E1 -16341.906,E2 -16341.906} C_VEL
LIN {X 0,Y 312.283,Z 254.83,A -85,B 0,C 180,E1 -16342.581,E2 -16342.581} C_VEL
LIN {X 0,Y 309.537,Z 260.52,A -85,B 0,C 180,E1 -16346.787,E2 -16346.787} C_VEL
LIN {X 0,Y 309.993,Z 262.405,A -85,B 0,C 180,E1 -16347.283,E2 -16347.283} C_VEL
LIN {X 0,Y 311.361,Z 265.487,A -85,B 0,C 180,E1 -16348.135,E2 -16348.135} C_VEL
LIN {X 0,Y 315.411,Z 277.293,A -85,B 0,C 180,E1 -16350.831,E2 -16350.831} C_VEL
LIN {X 0,Y 317.394,Z 284.81,A -85,B 0,C 180,E1 -16352.342,E2 -16352.342} C_VEL
LIN {X 0,Y 319.078,Z 295.118,A -85,B 0,C 180,E1 -16354.242,E2 -16354.242} C_VEL
LIN {X 0,Y 319.269,Z 298.861,A -85,B 0,C 180,E1 -16354.881,E2 -16354.881} C_VEL
LIN {X 0,Y 316.126,Z 310.785,A -85,B 0,C 180,E1 -16356.411,E2 -16356.411} C_VEL
LIN {X 0,Y 312.706,Z 322.112,A -85,B 0,C 180,E1 -16358.233,E2 -16358.233} C_VEL
LIN {X 0,Y 309.592,Z 331.372,A -85,B 0,C 180,E1 -16360.092,E2 -16360.092} C_VEL
LIN {X 0,Y 306.868,Z 339.004,A -85,B 0,C 180,E1 -16361.99,E2 -16361.99} C_VEL
LIN {X 0,Y 304.525,Z 345.292,A -85,B 0,C 180,E1 -16363.922,E2 -16363.922} C_VEL
LIN {X 0,Y 302.642,Z 350.379,A -85,B 0,C 180,E1 -16365.887,E2 -16365.887} C_VEL
LIN {X 0,Y 300.442,Z 355.53,A -85,B 0,C 180,E1 -16368.531,E2 -16368.531} C_VEL
LIN {X 0,Y 299.293,Z 358.253,A -85,B 0,C 180,E1 -16370.539,E2 -16370.539} C_VEL
LIN {X 0,Y 298.44,Z 359.613,A -85,B 0,C 180,E1 -16371.877,E2 -16371.877} C_VEL
LIN {X 0,Y 297.952,Z 360.536,A -85,B 0,C 180,E1 -16373.227,E2 -16373.227} C_VEL
LIN {X 0,Y 297.715,Z 361.032,A -85,B 0,C 180,E1 -16374.582,E2 -16374.582} C_VEL
LIN {X 0,Y 297.398,Z 361.169,A -85,B 0,C 180,E1 -16375.935,E2 -16375.935} C_VEL
LIN {X 0,Y 297.083,Z 360.927,A -85,B 0,C 180,E1 -16377.288,E2 -16377.288} C_VEL
LIN {X 0,Y 296.881,Z 360.266,A -85,B 0,C 180,E1 -16378.644,E2 -16378.644} C_VEL
LIN {X 0,Y 296.719,Z 357.703,A -85,B 0,C 180,E1 -16381.357,E2 -16381.357} C_VEL
LIN {X 0,Y 296.827,Z 354.673,A -85,B 0,C 180,E1 -16383.394,E2 -16383.394} C_VEL
LIN {X 0,Y 296.939,Z 350.599,A -85,B 0,C 180,E1 -16385.433,E2 -16385.433} C_VEL
LIN {X 0,Y 297.299,Z 344.388,A -85,B 0,C 180,E1 -16387.812,E2 -16387.812} C_VEL
LIN {X 0,Y 297.923,Z 336.396,A -85,B 0,C 180,E1 -16390.191,E2 -16390.191} C_VEL
LIN {X 0,Y 298.621,Z 327.748,A -85,B 0,C 180,E1 -16392.229,E2 -16392.229} C_VEL
LIN {X 0,Y 299.667,Z 317.128,A -85,B 0,C 180,E1 -16394.256,E2 -16394.256} C_VEL
LIN {X 0,Y 300.689,Z 306.159,A -85,B 0,C 180,E1 -16395.94,E2 -16395.94} C_VEL
LIN {X 0,Y 301.559,Z 294.873,A -85,B 0,C 180,E1 -16397.358,E2 -16397.358} C_VEL
LIN {X 0,Y 302.559,Z 282.098,A -85,B 0,C 180,E1 -16398.626,E2 -16398.626} C_VEL
LIN {X 0,Y 302.553,Z 278.012,A -85,B 0,C 180,E1 -16398.978,E2 -16398.978} C_VEL
LIN {X 0,Y 300.499,Z 264.916,A -85,B 0,C 180,E1 -16399.994,E2 -16399.994} C_VEL
LIN {X 0,Y 298.601,Z 251.678,A -85,B 0,C 180,E1 -16400.764,E2 -16400.764} C_VEL
LIN {X 0,Y 299.064,Z 242.219,A -85,B 0,C 180,E1 -16405.024,E2 -16405.024} C_VEL
LIN {X 0,Y 299.445,Z 234.013,A -85,B 0,C 180,E1 -16408.76,E2 -16408.76} C_VEL
LIN {X 0,Y 299.99,Z 225.618,A -85,B 0,C 180,E1 -16412.604,E2 -16412.604} C_VEL
LIN {X 0,Y 300.306,Z 218.707,A -85,B 0,C 180,E1 -16415.808,E2 -16415.808} C_VEL
LIN {X 0,Y 299.771,Z 213.322,A -85,B 0,C 180,E1 -16418.368,E2 -16418.368} C_VEL
LIN {X 0,Y 298.446,Z 206.311,A -85,B 0,C 180,E1 -16421.815,E2 -16421.815} C_VEL
LIN {X 0,Y 298.36,Z 206.317,A -85,B 0,C 180,E1 -16425.034,E2 -16425.034} C_VEL
LIN {X 0,Y 298.389,Z 206.317,A -85,B 0,C 180,E1 -16428.737,E2 -16428.737} C_VEL
LIN {X 0,Y 298.404,Z 206.318,A -85,B 0,C 180,E1 -16432.239,E2 -16432.239} C_VEL
LIN {X 0,Y 298.458,Z 206.489,A -85,B 0,C 180,E1 -16436.197,E2 -16436.197} C_VEL
LIN {X 0,Y 298.796,Z 209.048,A -85,B 0,C 180,E1 -16438.836,E2 -16438.836} C_VEL
LIN {X 0,Y 298.843,Z 212.236,A -85,B 0,C 180,E1 -16441.941,E2 -16441.941} C_VEL
LIN {X 0,Y 298.755,Z 215.512,A -85,B 0,C 180,E1 -16444.947,E2 -16444.947} C_VEL
LIN {X 0,Y 298.631,Z 218.821,A -85,B 0,C 180,E1 -16447.879,E2 -16447.879} C_VEL
LIN {X 0,Y 298.633,Z 222.236,A -85,B 0,C 180,E1 -16450.761,E2 -16450.761} C_VEL
LIN {X 0,Y 298.591,Z 225.626,A -85,B 0,C 180,E1 -16453.328,E2 -16453.328} C_VEL
LIN {X 0,Y 301.489,Z 235.731,A -85,B 0,C 180,E1 -16454.067,E2 -16454.067} C_VEL
LIN {X 0,Y 303.703,Z 245.015,A -85,B 0,C 180,E1 -16454.966,E2 -16454.966} C_VEL
LIN {X 0,Y 304.6,Z 250.255,A -85,B 0,C 180,E1 -16455.58,E2 -16455.58} C_VEL
LIN {X 0,Y 304.082,Z 257.089,A -85,B 0,C 180,E1 -16456.404,E2 -16456.404} C_VEL
LIN {X 0,Y 303.39,Z 264.077,A -85,B 0,C 180,E1 -16457.455,E2 -16457.455} C_VEL
LIN {X 0,Y 302.312,Z 271.836,A -85,B 0,C 180,E1 -16458.941,E2 -16458.941} C_VEL
LIN {X 0,Y 301.25,Z 278.313,A -85,B 0,C 180,E1 -16460.599,E2 -16460.599} C_VEL
LIN {X 0,Y 300.504,Z 282.337,A -85,B 0,C 180,E1 -16461.932,E2 -16461.932} C_VEL
LIN {X 0,Y 300.064,Z 286.779,A -85,B 0,C 180,E1 -16463.948,E2 -16463.948} C_VEL
LIN {X 0,Y 299.258,Z 289.798,A -85,B 0,C 180,E1 -16465.958,E2 -16465.958} C_VEL
LIN {X 0,Y 299.102,Z 291.061,A -85,B 0,C 180,E1 -16467.305,E2 -16467.305} C_VEL
LIN {X 0,Y 298.91,Z 291.827,A -85,B 0,C 180,E1 -16468.651,E2 -16468.651} C_VEL
LIN {X 0,Y 298.832,Z 292.095,A -85,B 0,C 180,E1 -16469.998,E2 -16469.998} C_VEL
LIN {X 0,Y 298.907,Z 291.864,A -85,B 0,C 180,E1 -16471.346,E2 -16471.346} C_VEL
LIN {X 0,Y 299.098,Z 291.147,A -85,B 0,C 180,E1 -16472.692,E2 -16472.692} C_VEL
LIN {X 0,Y 299.255,Z 289.937,A -85,B 0,C 180,E1 -16474.038,E2 -16474.038} C_VEL
LIN {X 0,Y 300.055,Z 287,A -85,B 0,C 180,E1 -16476.048,E2 -16476.048} C_VEL
LIN {X 0,Y 300.469,Z 282.647,A -85,B 0,C 180,E1 -16478.066,E2 -16478.066} C_VEL
LIN {X 0,Y 301.123,Z 279.743,A -85,B 0,C 180,E1 -16479.062,E2 -16479.062} C_VEL
LIN {X 0,Y 301.868,Z 275.049,A -85,B 0,C 180,E1 -16480.393,E2 -16480.393} C_VEL
LIN {X 0,Y 302.802,Z 269.165,A -85,B 0,C 180,E1 -16481.716,E2 -16481.716} C_VEL
LIN {X 0,Y 303.571,Z 262.755,A -85,B 0,C 180,E1 -16482.873,E2 -16482.873} C_VEL
LIN {X 0,Y 304.21,Z 255.525,A -85,B 0,C 180,E1 -16483.92,E2 -16483.92} C_VEL
LIN {X 0,Y 304.623,Z 250.349,A -85,B 0,C 180,E1 -16484.54,E2 -16484.54} C_VEL
LIN {X 0,Y 302.895,Z 241.127,A -85,B 0,C 180,E1 -16485.549,E2 -16485.549} C_VEL
LIN {X 0,Y 300.233,Z 230.903,A -85,B 0,C 180,E1 -16486.425,E2 -16486.425} C_VEL
LIN {X 0,Y 298.6,Z 225.424,A -85,B 0,C 180,E1 -16486.817,E2 -16486.817} C_VEL
LIN {X 0,Y 298.616,Z 220.68,A -85,B 0,C 180,E1 -16490.671,E2 -16490.671} C_VEL
LIN {X 0,Y 298.716,Z 217.312,A -85,B 0,C 180,E1 -16493.574,E2 -16493.574} C_VEL
LIN {X 0,Y 298.857,Z 213.876,A -85,B 0,C 180,E1 -16496.668,E2 -16496.668} C_VEL
LIN {X 0,Y 298.872,Z 210.815,A -85,B 0,C 180,E1 -16499.589,E2 -16499.589} C_VEL
LIN {X 0,Y 298.598,Z 207.642,A -85,B 0,C 180,E1 -16502.773,E2 -16502.773} C_VEL
LIN {X 0,Y 298.432,Z 206.313,A -85,B 0,C 180,E1 -16504.209,E2 -16504.209} C_VEL
LIN {X 0,Y 298.427,Z 206.312,A -85,B 0,C 180,E1 -16507.754,E2 -16507.754} C_VEL
LIN {X 0,Y 298.379,Z 206.317,A -85,B 0,C 180,E1 -16511.26,E2 -16511.26} C_VEL
LIN {X 0,Y 298.382,Z 206.319,A -85,B 0,C 180,E1 -16515.04,E2 -16515.04} C_VEL
LIN {X 0,Y 298.405,Z 206.312,A -85,B 0,C 180,E1 -16518.742,E2 -16518.742} C_VEL
LIN {X 0,Y 298.417,Z 206.309,A -85,B 0,C 180,E1 -16522.242,E2 -16522.242} C_VEL
LIN {X 0,Y 298.4,Z 206.312,A -85,B 0,C 180,E1 -16525.58,E2 -16525.58} C_VEL
LIN {X 0,Y 298.39,Z 206.315,A -85,B 0,C 180,E1 -16528.79,E2 -16528.79} C_VEL
LIN {X 0,Y 298.455,Z 206.306,A -85,B 0,C 180,E1 -16531.903,E2 -16531.903} C_VEL
LIN {X 0,Y 298.476,Z 206.294,A -85,B 0,C 180,E1 -16534.923,E2 -16534.923} C_VEL
LIN {X 0,Y 298.44,Z 206.301,A -85,B 0,C 180,E1 -16539.314,E2 -16539.314} C_VEL
LIN {X 0,Y 298.528,Z 206.3,A -85,B 0,C 180,E1 -16542.179,E2 -16542.179} C_VEL
LIN {X 0,Y 298.583,Z 206.279,A -85,B 0,C 180,E1 -16544.994,E2 -16544.994} C_VEL
LIN {X 0,Y 298.529,Z 206.295,A -85,B 0,C 180,E1 -16546.634,E2 -16546.634} C_VEL
LIN {X 0,Y 297.849,Z 206.383,A -85,B 0,C 180,E1 -16547.761,E2 -16547.761} C_VEL
LIN {X 0,Y 295.046,Z 206.724,A -85,B 0,C 180,E1 -16549.599,E2 -16549.599} C_VEL
LIN {X 0,Y 292.712,Z 207.015,A -85,B 0,C 180,E1 -16551.09,E2 -16551.09} C_VEL
LIN {X 0,Y 291.749,Z 207.141,A -85,B 0,C 180,E1 -16552.243,E2 -16552.243} C_VEL
LIN {X 0,Y 291.69,Z 207.147,A -85,B 0,C 180,E1 -16552.633,E2 -16552.633} C_VEL
LIN {X 0,Y 291.778,Z 207.139,A -85,B 0,C 180,E1 -16557.239,E2 -16557.239} C_VEL
LIN {X 0,Y 291.954,Z 207.104,A -85,B 0,C 180,E1 -16560,E2 -16560} C_VEL
LIN {X 0,Y 291.775,Z 207.141,A -85,B 0,C 180,E1 -16562.761,E2 -16562.761} C_VEL
LIN {X 0,Y 291.734,Z 207.147,A -85,B 0,C 180,E1 -16566.918,E2 -16566.918} C_VEL
LIN {X 0,Y 291.618,Z 207.15,A -85,B 0,C 180,E1 -16569.712,E2 -16569.712} C_VEL
LIN {X 0,Y 291.504,Z 207.165,A -85,B 0,C 180,E1 -16573.951,E2 -16573.951} C_VEL
LIN {X 0,Y 291.419,Z 207.179,A -85,B 0,C 180,E1 -16576.822,E2 -16576.822} C_VEL
LIN {X 0,Y 291.38,Z 207.193,A -85,B 0,C 180,E1 -16579.843,E2 -16579.843} C_VEL
LIN {X 0,Y 291.322,Z 207.198,A -85,B 0,C 180,E1 -16584.212,E2 -16584.212} C_VEL
LIN {X 0,Y 291.339,Z 207.197,A -85,B 0,C 180,E1 -16587.28,E2 -16587.28} C_VEL
LIN {X 0,Y 291.308,Z 207.199,A -85,B 0,C 180,E1 -16590.44,E2 -16590.44} C_VEL
LIN {X 0,Y 291.334,Z 207.193,A -85,B 0,C 180,E1 -16593.7,E2 -16593.7} C_VEL
LIN {X 0,Y 291.35,Z 207.191,A -85,B 0,C 180,E1 -16597.251,E2 -16597.251} C_VEL
LIN {X 0,Y 291.345,Z 207.206,A -85,B 0,C 180,E1 -16600.155,E2 -16600.155} C_VEL
LIN {X 0,Y 293.054,Z 214.394,A -85,B 0,C 180,E1 -16604.065,E2 -16604.065} C_VEL
LIN {X 0,Y 294.799,Z 221.674,A -85,B 0,C 180,E1 -16607.65,E2 -16607.65} C_VEL
LIN {X 0,Y 296.422,Z 228.794,A -85,B 0,C 180,E1 -16610.896,E2 -16610.896} C_VEL
LIN {X 0,Y 298.407,Z 238.007,A -85,B 0,C 180,E1 -16614.749,E2 -16614.749} C_VEL
LIN {X 0,Y 299.201,Z 242.394,A -85,B 0,C 180,E1 -16616.498,E2 -16616.498} C_VEL
LIN {X 0,Y 298.07,Z 247.739,A -85,B 0,C 180,E1 -16618.365,E2 -16618.365} C_VEL
LIN {X 0,Y 294.75,Z 262.311,A -85,B 0,C 180,E1 -16623.446,E2 -16623.446} C_VEL
LIN {X 0,Y 292.649,Z 273.569,A -85,B 0,C 180,E1 -16627.452,E2 -16627.452} C_VEL
LIN {X 0,Y 293.883,Z 287.171,A -85,B 0,C 180,E1 -16628.2,E2 -16628.2} C_VEL
LIN {X 0,Y 294.309,Z 300.363,A -85,B 0,C 180,E1 -16629.196,E2 -16629.196} C_VEL
LIN {X 0,Y 294.582,Z 311.435,A -85,B 0,C 180,E1 -16630.309,E2 -16630.309} C_VEL
LIN {X 0,Y 294.466,Z 321.556,A -85,B 0,C 180,E1 -16631.567,E2 -16631.567} C_VEL
LIN {X 0,Y 293.093,Z 333.751,A -85,B 0,C 180,E1 -16633.279,E2 -16633.279} C_VEL
LIN {X 0,Y 291.978,Z 345.643,A -85,B 0,C 180,E1 -16635.006,E2 -16635.006} C_VEL
LIN {X 0,Y 291.206,Z 355.281,A -85,B 0,C 180,E1 -16636.748,E2 -16636.748} C_VEL
LIN {X 0,Y 290.494,Z 364.705,A -85,B 0,C 180,E1 -16638.842,E2 -16638.842} C_VEL
LIN {X 0,Y 290.121,Z 372.243,A -85,B 0,C 180,E1 -16640.942,E2 -16640.942} C_VEL
LIN {X 0,Y 289.934,Z 378.259,A -85,B 0,C 180,E1 -16643.04,E2 -16643.04} C_VEL
LIN {X 0,Y 289.914,Z 382.976,A -85,B 0,C 180,E1 -16645.135,E2 -16645.135} C_VEL
LIN {X 0,Y 289.986,Z 386.511,A -85,B 0,C 180,E1 -16647.224,E2 -16647.224} C_VEL
LIN {X 0,Y 290.038,Z 388.272,A -85,B 0,C 180,E1 -16648.613,E2 -16648.613} C_VEL
LIN {X 0,Y 290.033,Z 389.535,A -85,B 0,C 180,E1 -16650.002,E2 -16650.002} C_VEL
LIN {X 0,Y 289.964,Z 390.361,A -85,B 0,C 180,E1 -16651.391,E2 -16651.391} C_VEL
LIN {X 0,Y 289.674,Z 390.762,A -85,B 0,C 180,E1 -16652.783,E2 -16652.783} C_VEL
LIN {X 0,Y 289.669,Z 390.773,A -85,B 0,C 180,E1 -16654.176,E2 -16654.176} C_VEL
LIN {X 0,Y 289.673,Z 389.507,A -85,B 0,C 180,E1 -16656.969,E2 -16656.969} C_VEL
LIN {X 0,Y 290.248,Z 386.699,A -85,B 0,C 180,E1 -16659.76,E2 -16659.76} C_VEL
LIN {X 0,Y 291.385,Z 382.227,A -85,B 0,C 180,E1 -16662.539,E2 -16662.539} C_VEL
LIN {X 0,Y 292.846,Z 377.767,A -85,B 0,C 180,E1 -16664.597,E2 -16664.597} C_VEL
LIN {X 0,Y 294.963,Z 371.244,A -85,B 0,C 180,E1 -16666.972,E2 -16666.972} C_VEL
LIN {X 0,Y 297.585,Z 363.127,A -85,B 0,C 180,E1 -16669.309,E2 -16669.309} C_VEL
LIN {X 0,Y 300.589,Z 354.647,A -85,B 0,C 180,E1 -16671.249,E2 -16671.249} C_VEL
LIN {X 0,Y 304.016,Z 344.511,A -85,B 0,C 180,E1 -16673.142,E2 -16673.142} C_VEL
LIN {X 0,Y 307.881,Z 332.215,A -85,B 0,C 180,E1 -16674.981,E2 -16674.981} C_VEL
LIN {X 0,Y 310.535,Z 320.254,A -85,B 0,C 180,E1 -16676.552,E2 -16676.552} C_VEL
LIN {X 0,Y 311.89,Z 309.116,A -85,B 0,C 180,E1 -16677.951,E2 -16677.951} C_VEL
LIN {X 0,Y 312.183,Z 297.764,A -85,B 0,C 180,E1 -16679.401,E2 -16679.401} C_VEL
LIN {X 0,Y 311.258,Z 284.755,A -85,B 0,C 180,E1 -16681.181,E2 -16681.181} C_VEL
LIN {X 0,Y 309.588,Z 273.466,A -85,B 0,C 180,E1 -16682.926,E2 -16682.926} C_VEL
LIN {X 0,Y 309.156,Z 269.913,A -85,B 0,C 180,E1 -16683.554,E2 -16683.554} C_VEL
LIN {X 0,Y 310.297,Z 265.647,A -85,B 0,C 180,E1 -16684.797,E2 -16684.797} C_VEL
LIN {X 0,Y 310.636,Z 263.805,A -85,B 0,C 180,E1 -16685.463,E2 -16685.463} C_VEL
LIN {X 0,Y 310.59,Z 259.603,A -85,B 0,C 180,E1 -16687.66,E2 -16687.66} C_VEL
LIN {X 0,Y 310.504,Z 256.843,A -85,B 0,C 180,E1 -16689.685,E2 -16689.685} C_VEL
LIN {X 0,Y 310.09,Z 255.33,A -85,B 0,C 180,E1 -16691.589,E2 -16691.589} C_VEL
LIN {X 0,Y 309.389,Z 254.766,A -85,B 0,C 180,E1 -16693.372,E2 -16693.372} C_VEL
LIN {X 0,Y 308.719,Z 254.704,A -85,B 0,C 180,E1 -16695.112,E2 -16695.112} C_VEL
LIN {X 0,Y 308.123,Z 255.028,A -85,B 0,C 180,E1 -16696.879,E2 -16696.879} C_VEL
LIN {X 0,Y 307.118,Z 256.645,A -85,B 0,C 180,E1 -16700.153,E2 -16700.153} C_VEL
LIN {X 0,Y 306.57,Z 257.892,A -85,B 0,C 180,E1 -16701.759,E2 -16701.759} C_VEL
LIN {X 0,Y 305.373,Z 260.024,A -85,B 0,C 180,E1 -16703.661,E2 -16703.661} C_VEL
LIN {X 0,Y 304.48,Z 261.716,A -85,B 0,C 180,E1 -16704.908,E2 -16704.908} C_VEL
LIN {X 0,Y 307.787,Z 271.136,A -85,B 0,C 180,E1 -16707.659,E2 -16707.659} C_VEL
LIN {X 0,Y 310.878,Z 281.451,A -85,B 0,C 180,E1 -16710.175,E2 -16710.175} C_VEL
LIN {X 0,Y 312.594,Z 289.17,A -85,B 0,C 180,E1 -16711.827,E2 -16711.827} C_VEL
LIN {X 0,Y 313.8,Z 299.486,A -85,B 0,C 180,E1 -16713.843,E2 -16713.843} C_VEL
LIN {X 0,Y 313.765,Z 301.668,A -85,B 0,C 180,E1 -16714.222,E2 -16714.222} C_VEL
LIN {X 0,Y 310.629,Z 312.268,A -85,B 0,C 180,E1 -16715.639,E2 -16715.639} C_VEL
LIN {X 0,Y 307.05,Z 323.223,A -85,B 0,C 180,E1 -16717.456,E2 -16717.456} C_VEL
LIN {X 0,Y 303.222,Z 333.677,A -85,B 0,C 180,E1 -16719.655,E2 -16719.655} C_VEL
LIN {X 0,Y 300.367,Z 340.949,A -85,B 0,C 180,E1 -16721.586,E2 -16721.586} C_VEL
LIN {X 0,Y 297.899,Z 346.914,A -85,B 0,C 180,E1 -16723.555,E2 -16723.555} C_VEL
LIN {X 0,Y 295.9,Z 351.746,A -85,B 0,C 180,E1 -16725.559,E2 -16725.559} C_VEL
LIN {X 0,Y 293.576,Z 356.653,A -85,B 0,C 180,E1 -16728.259,E2 -16728.259} C_VEL
LIN {X 0,Y 292.363,Z 359.181,A -85,B 0,C 180,E1 -16730.313,E2 -16730.313} C_VEL
LIN {X 0,Y 291.477,Z 360.402,A -85,B 0,C 180,E1 -16731.682,E2 -16731.682} C_VEL
LIN {X 0,Y 290.655,Z 361.6,A -85,B 0,C 180,E1 -16734.45,E2 -16734.45} C_VEL
LIN {X 0,Y 290.328,Z 361.646,A -85,B 0,C 180,E1 -16735.835,E2 -16735.835} C_VEL
LIN {X 0,Y 290,Z 361.274,A -85,B 0,C 180,E1 -16737.222,E2 -16737.222} C_VEL
LIN {X 0,Y 289.654,Z 359.329,A -85,B 0,C 180,E1 -16740,E2 -16740} C_VEL
LIN {X 0,Y 289.642,Z 356.789,A -85,B 0,C 180,E1 -16742.086,E2 -16742.086} C_VEL
LIN {X 0,Y 289.801,Z 353.256,A -85,B 0,C 180,E1 -16744.172,E2 -16744.172} C_VEL
LIN {X 0,Y 289.941,Z 348.398,A -85,B 0,C 180,E1 -16746.364,E2 -16746.364} C_VEL
LIN {X 0,Y 290.399,Z 341.722,A -85,B 0,C 180,E1 -16748.7,E2 -16748.7} C_VEL
LIN {X 0,Y 290.999,Z 334.253,A -85,B 0,C 180,E1 -16750.788,E2 -16750.788} C_VEL
LIN {X 0,Y 291.799,Z 325.07,A -85,B 0,C 180,E1 -16752.873,E2 -16752.873} C_VEL
LIN {X 0,Y 292.918,Z 313.713,A -85,B 0,C 180,E1 -16754.947,E2 -16754.947} C_VEL
LIN {X 0,Y 293.856,Z 303.167,A -85,B 0,C 180,E1 -16756.5,E2 -16756.5} C_VEL
LIN {X 0,Y 294.822,Z 291.662,A -85,B 0,C 180,E1 -16757.882,E2 -16757.882} C_VEL
LIN {X 0,Y 295.565,Z 279.144,A -85,B 0,C 180,E1 -16759.084,E2 -16759.084} C_VEL
LIN {X 0,Y 293.568,Z 266.309,A -85,B 0,C 180,E1 -16760.121,E2 -16760.121} C_VEL
LIN {X 0,Y 291.671,Z 252.941,A -85,B 0,C 180,E1 -16760.932,E2 -16760.932} C_VEL
LIN {X 0,Y 291.568,Z 251.982,A -85,B 0,C 180,E1 -16761.004,E2 -16761.004} C_VEL
LIN {X 0,Y 292.009,Z 243.424,A -85,B 0,C 180,E1 -16764.91,E2 -16764.91} C_VEL
LIN {X 0,Y 292.4,Z 235.133,A -85,B 0,C 180,E1 -16768.732,E2 -16768.732} C_VEL
LIN {X 0,Y 292.995,Z 226.128,A -85,B 0,C 180,E1 -16772.906,E2 -16772.906} C_VEL
LIN {X 0,Y 293.294,Z 219.427,A -85,B 0,C 180,E1 -16776.044,E2 -16776.044} C_VEL
LIN {X 0,Y 292.704,Z 214.093,A -85,B 0,C 180,E1 -16778.629,E2 -16778.629} C_VEL
LIN {X 0,Y 291.394,Z 207.189,A -85,B 0,C 180,E1 -16782.118,E2 -16782.118} C_VEL
LIN {X 0,Y 291.315,Z 207.198,A -85,B 0,C 180,E1 -16786.365,E2 -16786.365} C_VEL
LIN {X 0,Y 291.382,Z 207.191,A -85,B 0,C 180,E1 -16790.518,E2 -16790.518} C_VEL
LIN {X 0,Y 291.396,Z 207.192,A -85,B 0,C 180,E1 -16792.916,E2 -16792.916} C_VEL
LIN {X 0,Y 291.389,Z 207.262,A -85,B 0,C 180,E1 -16795.498,E2 -16795.498} C_VEL
LIN {X 0,Y 291.786,Z 209.635,A -85,B 0,C 180,E1 -16798,E2 -16798} C_VEL
LIN {X 0,Y 291.868,Z 212.876,A -85,B 0,C 180,E1 -16801.209,E2 -16801.209} C_VEL
LIN {X 0,Y 291.802,Z 216.132,A -85,B 0,C 180,E1 -16804.307,E2 -16804.307} C_VEL
LIN {X 0,Y 291.661,Z 219.5,A -85,B 0,C 180,E1 -16807.321,E2 -16807.321} C_VEL
LIN {X 0,Y 291.641,Z 222.936,A -85,B 0,C 180,E1 -16810.281,E2 -16810.281} C_VEL
LIN {X 0,Y 291.562,Z 226.069,A -85,B 0,C 180,E1 -16812.824,E2 -16812.824} C_VEL
LIN {X 0,Y 294.762,Z 237.092,A -85,B 0,C 180,E1 -16813.675,E2 -16813.675} C_VEL
LIN {X 0,Y 296.937,Z 246.426,A -85,B 0,C 180,E1 -16814.619,E2 -16814.619} C_VEL
LIN {X 0,Y 297.806,Z 251.471,A -85,B 0,C 180,E1 -16815.238,E2 -16815.238} C_VEL
LIN {X 0,Y 297.119,Z 259.95,A -85,B 0,C 180,E1 -16816.316,E2 -16816.316} C_VEL
LIN {X 0,Y 296.203,Z 267.978,A -85,B 0,C 180,E1 -16817.668,E2 -16817.668} C_VEL
LIN {X 0,Y 295.193,Z 274.309,A -85,B 0,C 180,E1 -16819.018,E2 -16819.018} C_VEL
LIN {X 0,Y 294.319,Z 279.325,A -85,B 0,C 180,E1 -16820.376,E2 -16820.376} C_VEL
LIN {X 0,Y 293.546,Z 283.332,A -85,B 0,C 180,E1 -16821.739,E2 -16821.739} C_VEL
LIN {X 0,Y 293.077,Z 287.763,A -85,B 0,C 180,E1 -16823.803,E2 -16823.803} C_VEL
LIN {X 0,Y 292.249,Z 290.773,A -85,B 0,C 180,E1 -16825.861,E2 -16825.861} C_VEL
LIN {X 0,Y 292.083,Z 292.035,A -85,B 0,C 180,E1 -16827.24,E2 -16827.24} C_VEL
LIN {X 0,Y 291.884,Z 292.801,A -85,B 0,C 180,E1 -16828.619,E2 -16828.619} C_VEL
LIN {X 0,Y 291.804,Z 293.069,A -85,B 0,C 180,E1 -16829.998,E2 -16829.998} C_VEL
LIN {X 0,Y 291.882,Z 292.837,A -85,B 0,C 180,E1 -16831.378,E2 -16831.378} C_VEL
LIN {X 0,Y 292.079,Z 292.121,A -85,B 0,C 180,E1 -16832.757,E2 -16832.757} C_VEL
LIN {X 0,Y 292.246,Z 290.912,A -85,B 0,C 180,E1 -16834.135,E2 -16834.135} C_VEL
LIN {X 0,Y 293.067,Z 287.979,A -85,B 0,C 180,E1 -16836.193,E2 -16836.193} C_VEL
LIN {X 0,Y 293.51,Z 283.635,A -85,B 0,C 180,E1 -16838.258,E2 -16838.258} C_VEL
LIN {X 0,Y 294.185,Z 280.745,A -85,B 0,C 180,E1 -16839.278,E2 -16839.278} C_VEL
LIN {X 0,Y 294.952,Z 276.076,A -85,B 0,C 180,E1 -16840.64,E2 -16840.64} C_VEL
LIN {X 0,Y 295.937,Z 270.221,A -85,B 0,C 180,E1 -16841.991,E2 -16841.991} C_VEL
LIN {X 0,Y 296.738,Z 263.854,A -85,B 0,C 180,E1 -16843.175,E2 -16843.175} C_VEL
LIN {X 0,Y 297.4,Z 256.648,A -85,B 0,C 180,E1 -16844.251,E2 -16844.251} C_VEL
LIN {X 0,Y 297.857,Z 251.663,A -85,B 0,C 180,E1 -16844.867,E2 -16844.867} C_VEL
LIN {X 0,Y 296.17,Z 242.67,A -85,B 0,C 180,E1 -16845.902,E2 -16845.902} C_VEL
LIN {X 0,Y 293.407,Z 232.064,A -85,B 0,C 180,E1 -16846.859,E2 -16846.859} C_VEL
LIN {X 0,Y 291.563,Z 226.056,A -85,B 0,C 180,E1 -16847.319,E2 -16847.319} C_VEL
LIN {X 0,Y 291.649,Z 221.363,A -85,B 0,C 180,E1 -16851.188,E2 -16851.188} C_VEL
LIN {X 0,Y 291.751,Z 217.956,A -85,B 0,C 180,E1 -16854.172,E2 -16854.172} C_VEL
LIN {X 0,Y 291.865,Z 214.644,A -85,B 0,C 180,E1 -16857.224,E2 -16857.224} C_VEL
LIN {X 0,Y 291.847,Z 211.405,A -85,B 0,C 180,E1 -16860.376,E2 -16860.376} C_VEL
LIN {X 0,Y 291.557,Z 208.186,A -85,B 0,C 180,E1 -16863.668,E2 -16863.668} C_VEL
LIN {X 0,Y 291.385,Z 207.19,A -85,B 0,C 180,E1 -16864.909,E2 -16864.909} C_VEL
LIN {X 0,Y 291.39,Z 207.191,A -85,B 0,C 180,E1 -16867.257,E2 -16867.257} C_VEL
LIN {X 0,Y 291.329,Z 207.197,A -85,B 0,C 180,E1 -16870.64,E2 -16870.64} C_VEL
LIN {X 0,Y 291.307,Z 207.196,A -85,B 0,C 180,E1 -16874.396,E2 -16874.396} C_VEL
LIN {X 0,Y 291.344,Z 207.195,A -85,B 0,C 180,E1 -16878.397,E2 -16878.397} C_VEL
LIN {X 0,Y 291.356,Z 207.193,A -85,B 0,C 180,E1 -16881.158,E2 -16881.158} C_VEL
LIN {X 0,Y 291.353,Z 207.194,A -85,B 0,C 180,E1 -16884.625,E2 -16884.625} C_VEL
LIN {X 0,Y 291.367,Z 207.19,A -85,B 0,C 180,E1 -16887.95,E2 -16887.95} C_VEL
LIN {X 0,Y 291.374,Z 207.184,A -85,B 0,C 180,E1 -16891.157,E2 -16891.157} C_VEL
LIN {X 0,Y 291.407,Z 207.177,A -85,B 0,C 180,E1 -16894.271,E2 -16894.271} C_VEL
LIN {X 0,Y 291.372,Z 207.19,A -85,B 0,C 180,E1 -16897.299,E2 -16897.299} C_VEL
LIN {X 0,Y 291.448,Z 207.171,A -85,B 0,C 180,E1 -16900.269,E2 -16900.269} C_VEL
LIN {X 0,Y 291.545,Z 207.155,A -85,B 0,C 180,E1 -16904.623,E2 -16904.623} C_VEL
LIN {X 0,Y 291.525,Z 207.165,A -85,B 0,C 180,E1 -16908.88,E2 -16908.88} C_VEL
LIN {X 0,Y 291.677,Z 207.149,A -85,B 0,C 180,E1 -16911.687,E2 -16911.687} C_VEL
LIN {X 0,Y 291.69,Z 207.147,A -85,B 0,C 180,E1 -16912.633,E2 -16912.633} C_VEL
LIN {X 0,Y 291.089,Z 207.228,A -85,B 0,C 180,E1 -16913.784,E2 -16913.784} C_VEL
LIN {X 0,Y 288.319,Z 207.581,A -85,B 0,C 180,E1 -16915.66,E2 -16915.66} C_VEL
LIN {X 0,Y 285.941,Z 207.875,A -85,B 0,C 180,E1 -16917.182,E2 -16917.182} C_VEL
LIN {X 0,Y 284.923,Z 207.992,A -85,B 0,C 180,E1 -16918.361,E2 -16918.361} C_VEL
LIN {X 0,Y 284.844,Z 207.997,A -85,B 0,C 180,E1 -16918.76,E2 -16918.76} C_VEL
LIN {X 0,Y 284.844,Z 207.999,A -85,B 0,C 180,E1 -16921.414,E2 -16921.414} C_VEL
LIN {X 0,Y 284.687,Z 208.024,A -85,B 0,C 180,E1 -16927.09,E2 -16927.09} C_VEL
